LIN {X 0,Y 591.929,Z 246.123,A -85,B 0,C 180,E1 27050.152,E2 27050.152} C_VEL
LIN {X 0,Y 584.236,Z 228.435,A -85,B 0,C 180,E1 27048.26,E2 27048.26} C_VEL
LIN {X 0,Y 578.995,Z 217.335,A -85,B 0,C 180,E1 27047.073,E2 27047.073} C_VEL
LIN {X 0,Y 577.607,Z 214.744,A -85,B 0,C 180,E1 27046.785,E2 27046.785} C_VEL
LIN {X 0,Y 577.299,Z 213.311,A -85,B 0,C 180,E1 27046.634,E2 27046.634} C_VEL
LIN {X 0,Y 577.308,Z 213.309,A -85,B 0,C 180,E1 27043.304,E2 27043.304} C_VEL
LIN {X 0,Y 577.314,Z 213.308,A -85,B 0,C 180,E1 27040.046,E2 27040.046} C_VEL
LIN {X 0,Y 577.298,Z 213.305,A -85,B 0,C 180,E1 27036.818,E2 27036.818} C_VEL
LIN {X 0,Y 577.315,Z 213.304,A -85,B 0,C 180,E1 27033.539,E2 27033.539} C_VEL
LIN {X 0,Y 577.32,Z 213.314,A -85,B 0,C 180,E1 27030.15,E2 27030.15} C_VEL
LIN {X 0,Y 577.304,Z 213.311,A -85,B 0,C 180,E1 27026.876,E2 27026.876} C_VEL
LIN {X 0,Y 577.307,Z 213.291,A -85,B 0,C 180,E1 27023.584,E2 27023.584} C_VEL
LIN {X 0,Y 577.316,Z 213.314,A -85,B 0,C 180,E1 27020.267,E2 27020.267} C_VEL
LIN {X 0,Y 577.309,Z 213.299,A -85,B 0,C 180,E1 27016.916,E2 27016.916} C_VEL
LIN {X 0,Y 577.3,Z 213.303,A -85,B 0,C 180,E1 27013.674,E2 27013.674} C_VEL
LIN {X 0,Y 577.315,Z 213.307,A -85,B 0,C 180,E1 27010.341,E2 27010.341} C_VEL
LIN {X 0,Y 577.319,Z 213.3,A -85,B 0,C 180,E1 27006.964,E2 27006.964} C_VEL
LIN {X 0,Y 577.297,Z 213.318,A -85,B 0,C 180,E1 27003.674,E2 27003.674} C_VEL
LIN {X 0,Y 577.313,Z 213.295,A -85,B 0,C 180,E1 27000.397,E2 27000.397} C_VEL
LIN {X 0,Y 577.307,Z 213.312,A -85,B 0,C 180,E1 26997.121,E2 26997.121} C_VEL
LIN {X 0,Y 577.294,Z 213.294,A -85,B 0,C 180,E1 26993.818,E2 26993.818} C_VEL
LIN {X 0,Y 577.317,Z 213.31,A -85,B 0,C 180,E1 26990.53,E2 26990.53} C_VEL
LIN {X 0,Y 577.291,Z 213.316,A -85,B 0,C 180,E1 26987.293,E2 26987.293} C_VEL
LIN {X 0,Y 577.307,Z 213.316,A -85,B 0,C 180,E1 26983.999,E2 26983.999} C_VEL
LIN {X 0,Y 577.319,Z 213.312,A -85,B 0,C 180,E1 26980.682,E2 26980.682} C_VEL
LIN {X 0,Y 577.283,Z 213.322,A -85,B 0,C 180,E1 26977.494,E2 26977.494} C_VEL
LIN {X 0,Y 577.32,Z 213.321,A -85,B 0,C 180,E1 26974.232,E2 26974.232} C_VEL
LIN {X 0,Y 577.294,Z 213.316,A -85,B 0,C 180,E1 26970.989,E2 26970.989} C_VEL
LIN {X 0,Y 577.282,Z 213.322,A -85,B 0,C 180,E1 26967.642,E2 26967.642} C_VEL
LIN {X 0,Y 577.322,Z 213.313,A -85,B 0,C 180,E1 26964.413,E2 26964.413} C_VEL
LIN {X 0,Y 577.271,Z 213.322,A -85,B 0,C 180,E1 26961.21,E2 26961.21} C_VEL
LIN {X 0,Y 577.318,Z 213.515,A -85,B 0,C 180,E1 26960.825,E2 26960.825} C_VEL
LIN {X 0,Y 578.825,Z 217.068,A -85,B 0,C 180,E1 26960.399,E2 26960.399} C_VEL
LIN {X 0,Y 588.305,Z 235.653,A -85,B 0,C 180,E1 26958.091,E2 26958.091} C_VEL
LIN {X 0,Y 600.676,Z 260.638,A -85,B 0,C 180,E1 26955.24,E2 26955.24} C_VEL
LIN {X 0,Y 607.806,Z 275.644,A -85,B 0,C 180,E1 26953.662,E2 26953.662} C_VEL
LIN {X 0,Y 605.103,Z 308.798,A -85,B 0,C 180,E1 26951.828,E2 26951.828} C_VEL
LIN {X 0,Y 607.828,Z 331.376,A -85,B 0,C 180,E1 26951.271,E2 26951.271} C_VEL
LIN {X 0,Y 602.232,Z 577.23,A -85,B 0,C 180,E1 26947.881,E2 26947.881} C_VEL
LIN {X 0,Y 599.928,Z 692.589,A -85,B 0,C 180,E1 26946.326,E2 26946.326} C_VEL
LIN {X 0,Y 598.876,Z 717.126,A -85,B 0,C 180,E1 26945.833,E2 26945.833} C_VEL
LIN {X 0,Y 597.663,Z 738.821,A -85,B 0,C 180,E1 26945.256,E2 26945.256} C_VEL
LIN {X 0,Y 596.011,Z 763.246,A -85,B 0,C 180,E1 26944.428,E2 26944.428} C_VEL
LIN {X 0,Y 594.427,Z 783.289,A -85,B 0,C 180,E1 26943.601,E2 26943.601} C_VEL
LIN {X 0,Y 592.413,Z 806.84,A -85,B 0,C 180,E1 26942.444,E2 26942.444} C_VEL
LIN {X 0,Y 590.599,Z 826.305,A -85,B 0,C 180,E1 26941.316,E2 26941.316} C_VEL
LIN {X 0,Y 588.459,Z 848.134,A -85,B 0,C 180,E1 26939.858,E2 26939.858} C_VEL
LIN {X 0,Y 586.519,Z 867.008,A -85,B 0,C 180,E1 26938.397,E2 26938.397} C_VEL
LIN {X 0,Y 584.495,Z 887.006,A -85,B 0,C 180,E1 26936.628,E2 26936.628} C_VEL
LIN {X 0,Y 582.762,Z 903.916,A -85,B 0,C 180,E1 26934.912,E2 26934.912} C_VEL
LIN {X 0,Y 581.074,Z 921.418,A -85,B 0,C 180,E1 26932.886,E2 26932.886} C_VEL
LIN {X 0,Y 579.75,Z 935.465,A -85,B 0,C 180,E1 26931.023,E2 26931.023} C_VEL
LIN {X 0,Y 578.56,Z 949.769,A -85,B 0,C 180,E1 26928.855,E2 26928.855} C_VEL
LIN {X 0,Y 577.681,Z 961.419,A -85,B 0,C 180,E1 26926.801,E2 26926.801} C_VEL
LIN {X 0,Y 576.975,Z 972.466,A -85,B 0,C 180,E1 26924.553,E2 26924.553} C_VEL
LIN {X 0,Y 576.545,Z 980.188,A -85,B 0,C 180,E1 26922.622,E2 26922.622} C_VEL
LIN {X 0,Y 576.225,Z 987.119,A -85,B 0,C 180,E1 26920.498,E2 26920.498} C_VEL
LIN {X 0,Y 576.012,Z 993.449,A -85,B 0,C 180,E1 26918.083,E2 26918.083} C_VEL
LIN {X 0,Y 575.941,Z 997.697,A -85,B 0,C 180,E1 26915.852,E2 26915.852} C_VEL
LIN {X 0,Y 575.915,Z 1000.576,A -85,B 0,C 180,E1 26913.683,E2 26913.683} C_VEL
LIN {X 0,Y 575.907,Z 1002.235,A -85,B 0,C 180,E1 26911.194,E2 26911.194} C_VEL
LIN {X 0,Y 575.888,Z 1002.325,A -85,B 0,C 180,E1 26909.204,E2 26909.204} C_VEL
LIN {X 0,Y 575.886,Z 1001.289,A -85,B 0,C 180,E1 26907.114,E2 26907.114} C_VEL
LIN {X 0,Y 575.909,Z 998.45,A -85,B 0,C 180,E1 26904.62,E2 26904.62} C_VEL
LIN {X 0,Y 575.969,Z 994.688,A -85,B 0,C 180,E1 26902.519,E2 26902.519} C_VEL
LIN {X 0,Y 576.141,Z 989.457,A -85,B 0,C 180,E1 26900.308,E2 26900.308} C_VEL
LIN {X 0,Y 576.451,Z 981.951,A -85,B 0,C 180,E1 26897.884,E2 26897.884} C_VEL
LIN {X 0,Y 576.79,Z 975.298,A -85,B 0,C 180,E1 26896.117,E2 26896.117} C_VEL
LIN {X 0,Y 577.322,Z 966.57,A -85,B 0,C 180,E1 26894.222,E2 26894.222} C_VEL
LIN {X 0,Y 578.171,Z 954.305,A -85,B 0,C 180,E1 26891.967,E2 26891.967} C_VEL
LIN {X 0,Y 579.14,Z 941.931,A -85,B 0,C 180,E1 26890.01,E2 26890.01} C_VEL
LIN {X 0,Y 580.46,Z 926.019,A -85,B 0,C 180,E1 26887.837,E2 26887.837} C_VEL
LIN {X 0,Y 581.785,Z 911.136,A -85,B 0,C 180,E1 26886.071,E2 26886.071} C_VEL
LIN {X 0,Y 583.484,Z 892.287,A -85,B 0,C 180,E1 26884.115,E2 26884.115} C_VEL
LIN {X 0,Y 585.062,Z 875.137,A -85,B 0,C 180,E1 26882.568,E2 26882.568} C_VEL
LIN {X 0,Y 586.934,Z 854.247,A -85,B 0,C 180,E1 26880.92,E2 26880.92} C_VEL
LIN {X 0,Y 588.596,Z 834.717,A -85,B 0,C 180,E1 26879.587,E2 26879.587} C_VEL
LIN {X 0,Y 590.519,Z 811.335,A -85,B 0,C 180,E1 26878.213,E2 26878.213} C_VEL
LIN {X 0,Y 592.038,Z 790.551,A -85,B 0,C 180,E1 26877.171,E2 26877.171} C_VEL
LIN {X 0,Y 593.635,Z 766.597,A -85,B 0,C 180,E1 26876.168,E2 26876.168} C_VEL
LIN {X 0,Y 594.899,Z 744.933,A -85,B 0,C 180,E1 26875.42,E2 26875.42} C_VEL
LIN {X 0,Y 596.12,Z 719.728,A -85,B 0,C 180,E1 26874.739,E2 26874.739} C_VEL
LIN {X 0,Y 596.892,Z 698.83,A -85,B 0,C 180,E1 26874.312,E2 26874.312} C_VEL
LIN {X 0,Y 597.508,Z 665.557,A -85,B 0,C 180,E1 26873.847,E2 26873.847} C_VEL
LIN {X 0,Y 599.383,Z 523.368,A -85,B 0,C 180,E1 26872.041,E2 26872.041} C_VEL
LIN {X 0,Y 602.037,Z 398.059,A -85,B 0,C 180,E1 26870.281,E2 26870.281} C_VEL
LIN {X 0,Y 603.978,Z 328.15,A -85,B 0,C 180,E1 26869.204,E2 26869.204} C_VEL
LIN {X 0,Y 603.753,Z 324.587,A -85,B 0,C 180,E1 26869.08,E2 26869.08} C_VEL
LIN {X 0,Y 608.265,Z 300.685,A -85,B 0,C 180,E1 26867.429,E2 26867.429} C_VEL
LIN {X 0,Y 613.531,Z 280.646,A -85,B 0,C 180,E1 26865.901,E2 26865.901} C_VEL
LIN {X 0,Y 612.091,Z 275.219,A -85,B 0,C 180,E1 26864.716,E2 26864.716} C_VEL
LIN {X 0,Y 611.11,Z 271.585,A -85,B 0,C 180,E1 26863.538,E2 26863.538} C_VEL
LIN {X 0,Y 610.691,Z 269.324,A -85,B 0,C 180,E1 26862.123,E2 26862.123} C_VEL
LIN {X 0,Y 610.625,Z 269.272,A -85,B 0,C 180,E1 26861.543,E2 26861.543} C_VEL
LIN {X 0,Y 610.726,Z 271.372,A -85,B 0,C 180,E1 26860.048,E2 26860.048} C_VEL
LIN {X 0,Y 611.329,Z 275.332,A -85,B 0,C 180,E1 26858.788,E2 26858.788} C_VEL
LIN {X 0,Y 611.672,Z 278.803,A -85,B 0,C 180,E1 26858.045,E2 26858.045} C_VEL
LIN {X 0,Y 605.574,Z 300.252,A -85,B 0,C 180,E1 26856.119,E2 26856.119} C_VEL
LIN {X 0,Y 599.965,Z 327.92,A -85,B 0,C 180,E1 26853.824,E2 26853.824} C_VEL
LIN {X 0,Y 595.013,Z 362.924,A -85,B 0,C 180,E1 26851.114,E2 26851.114} C_VEL
LIN {X 0,Y 590.47,Z 407.602,A -85,B 0,C 180,E1 26847.878,E2 26847.878} C_VEL
LIN {X 0,Y 589.4,Z 422.994,A -85,B 0,C 180,E1 26846.832,E2 26846.832} C_VEL
LIN {X 0,Y 592.686,Z 455.008,A -85,B 0,C 180,E1 26845.661,E2 26845.661} C_VEL
LIN {X 0,Y 595.543,Z 491.146,A -85,B 0,C 180,E1 26844.524,E2 26844.524} C_VEL
LIN {X 0,Y 594.867,Z 505.645,A -85,B 0,C 180,E1 26844.22,E2 26844.22} C_VEL
LIN {X 0,Y 589.455,Z 607.464,A -85,B 0,C 180,E1 26842.27,E2 26842.27} C_VEL
LIN {X 0,Y 586.293,Z 687.572,A -85,B 0,C 180,E1 26840.777,E2 26840.777} C_VEL
LIN {X 0,Y 585.33,Z 709.905,A -85,B 0,C 180,E1 26840.167,E2 26840.167} C_VEL
LIN {X 0,Y 584.359,Z 731.272,A -85,B 0,C 180,E1 26839.387,E2 26839.387} C_VEL
LIN {X 0,Y 583.386,Z 750.706,A -85,B 0,C 180,E1 26838.486,E2 26838.486} C_VEL
LIN {X 0,Y 582.433,Z 769.003,A -85,B 0,C 180,E1 26837.432,E2 26837.432} C_VEL
LIN {X 0,Y 581.473,Z 786.178,A -85,B 0,C 180,E1 26836.226,E2 26836.226} C_VEL
LIN {X 0,Y 580.594,Z 801.262,A -85,B 0,C 180,E1 26834.951,E2 26834.951} C_VEL
LIN {X 0,Y 579.773,Z 814.876,A -85,B 0,C 180,E1 26833.565,E2 26833.565} C_VEL
LIN {X 0,Y 579.038,Z 827.147,A -85,B 0,C 180,E1 26832.061,E2 26832.061} C_VEL
LIN {X 0,Y 578.439,Z 837.273,A -85,B 0,C 180,E1 26830.558,E2 26830.558} C_VEL
LIN {X 0,Y 577.896,Z 846.496,A -85,B 0,C 180,E1 26828.858,E2 26828.858} C_VEL
LIN {X 0,Y 577.499,Z 853.707,A -85,B 0,C 180,E1 26827.161,E2 26827.161} C_VEL
LIN {X 0,Y 577.21,Z 859.389,A -85,B 0,C 180,E1 26825.368,E2 26825.368} C_VEL
LIN {X 0,Y 576.993,Z 863.232,A -85,B 0,C 180,E1 26823.577,E2 26823.577} C_VEL
LIN {X 0,Y 576.852,Z 865.342,A -85,B 0,C 180,E1 26821.788,E2 26821.788} C_VEL
LIN {X 0,Y 576.771,Z 865.736,A -85,B 0,C 180,E1 26819.901,E2 26819.901} C_VEL
LIN {X 0,Y 576.736,Z 864.293,A -85,B 0,C 180,E1 26818.013,E2 26818.013} C_VEL
LIN {X 0,Y 576.764,Z 861.014,A -85,B 0,C 180,E1 26816.123,E2 26816.123} C_VEL
LIN {X 0,Y 576.874,Z 856.161,A -85,B 0,C 180,E1 26814.33,E2 26814.33} C_VEL
LIN {X 0,Y 577.061,Z 849.471,A -85,B 0,C 180,E1 26812.533,E2 26812.533} C_VEL
LIN {X 0,Y 577.367,Z 841.126,A -85,B 0,C 180,E1 26810.799,E2 26810.799} C_VEL
LIN {X 0,Y 577.814,Z 831.101,A -85,B 0,C 180,E1 26809.128,E2 26809.128} C_VEL
LIN {X 0,Y 578.397,Z 819.329,A -85,B 0,C 180,E1 26807.52,E2 26807.52} C_VEL
LIN {X 0,Y 579.11,Z 805.98,A -85,B 0,C 180,E1 26806.012,E2 26806.012} C_VEL
LIN {X 0,Y 579.937,Z 790.987,A -85,B 0,C 180,E1 26804.602,E2 26804.602} C_VEL
LIN {X 0,Y 580.827,Z 774.875,A -85,B 0,C 180,E1 26803.344,E2 26803.344} C_VEL
LIN {X 0,Y 581.733,Z 757.436,A -85,B 0,C 180,E1 26802.218,E2 26802.218} C_VEL
LIN {X 0,Y 582.635,Z 739.626,A -85,B 0,C 180,E1 26801.281,E2 26801.281} C_VEL
LIN {X 0,Y 583.514,Z 720.275,A -85,B 0,C 180,E1 26800.469,E2 26800.469} C_VEL
LIN {X 0,Y 584.279,Z 700.12,A -85,B 0,C 180,E1 26799.828,E2 26799.828} C_VEL
LIN {X 0,Y 584.919,Z 679.428,A -85,B 0,C 180,E1 26799.37,E2 26799.37} C_VEL
LIN {X 0,Y 588.981,Z 489.215,A -85,B 0,C 180,E1 26796.534,E2 26796.534} C_VEL
LIN {X 0,Y 585.221,Z 455.543,A -85,B 0,C 180,E1 26795.791,E2 26795.791} C_VEL
LIN {X 0,Y 587.587,Z 405.605,A -85,B 0,C 180,E1 26792.594,E2 26792.594} C_VEL
LIN {X 0,Y 590.441,Z 352.546,A -85,B 0,C 180,E1 26789.158,E2 26789.158} C_VEL
LIN {X 0,Y 593.46,Z 300.77,A -85,B 0,C 180,E1 26785.754,E2 26785.754} C_VEL
LIN {X 0,Y 595.914,Z 261.134,A -85,B 0,C 180,E1 26783.108,E2 26783.108} C_VEL
LIN {X 0,Y 591.877,Z 250.242,A -85,B 0,C 180,E1 26782.056,E2 26782.056} C_VEL
LIN {X 0,Y 589.101,Z 245.546,A -85,B 0,C 180,E1 26781.522,E2 26781.522} C_VEL
LIN {X 0,Y 577.793,Z 233.961,A -85,B 0,C 180,E1 26779.852,E2 26779.852} C_VEL
LIN {X 0,Y 576.198,Z 231.311,A -85,B 0,C 180,E1 26779.532,E2 26779.532} C_VEL
LIN {X 0,Y 569.344,Z 214.421,A -85,B 0,C 180,E1 26777.698,E2 26777.698} C_VEL
LIN {X 0,Y 569.381,Z 214.302,A -85,B 0,C 180,E1 26774.482,E2 26774.482} C_VEL
LIN {X 0,Y 569.39,Z 214.435,A -85,B 0,C 180,E1 26773.881,E2 26773.881} C_VEL
LIN {X 0,Y 570.341,Z 217.235,A -85,B 0,C 180,E1 26773.61,E2 26773.61} C_VEL
LIN {X 0,Y 571.71,Z 219.791,A -85,B 0,C 180,E1 26773.317,E2 26773.317} C_VEL
LIN {X 0,Y 578.876,Z 234.711,A -85,B 0,C 180,E1 26771.683,E2 26771.683} C_VEL
LIN {X 0,Y 586.838,Z 253.704,A -85,B 0,C 180,E1 26769.633,E2 26769.633} C_VEL
LIN {X 0,Y 593.746,Z 272.147,A -85,B 0,C 180,E1 26767.674,E2 26767.674} C_VEL
LIN {X 0,Y 592.76,Z 314.667,A -85,B 0,C 180,E1 26764.643,E2 26764.643} C_VEL
LIN {X 0,Y 592.824,Z 338.961,A -85,B 0,C 180,E1 26763.068,E2 26763.068} C_VEL
LIN {X 0,Y 591.933,Z 343.747,A -85,B 0,C 180,E1 26762.899,E2 26762.899} C_VEL
LIN {X 0,Y 589.728,Z 439.794,A -85,B 0,C 180,E1 26761.581,E2 26761.581} C_VEL
LIN {X 0,Y 586.74,Z 530.066,A -85,B 0,C 180,E1 26760.163,E2 26760.163} C_VEL
LIN {X 0,Y 583.259,Z 625.148,A -85,B 0,C 180,E1 26758.492,E2 26758.492} C_VEL
LIN {X 0,Y 582.489,Z 647.168,A -85,B 0,C 180,E1 26757.952,E2 26757.952} C_VEL
LIN {X 0,Y 581.453,Z 668.771,A -85,B 0,C 180,E1 26757.245,E2 26757.245} C_VEL
LIN {X 0,Y 580.207,Z 690.159,A -85,B 0,C 180,E1 26756.345,E2 26756.345} C_VEL
LIN {X 0,Y 578.823,Z 710.131,A -85,B 0,C 180,E1 26755.312,E2 26755.312} C_VEL
LIN {X 0,Y 577.378,Z 729.317,A -85,B 0,C 180,E1 26754.123,E2 26754.123} C_VEL
LIN {X 0,Y 575.82,Z 748.322,A -85,B 0,C 180,E1 26752.728,E2 26752.728} C_VEL
LIN {X 0,Y 574.417,Z 765.121,A -85,B 0,C 180,E1 26751.281,E2 26751.281} C_VEL
LIN {X 0,Y 573.057,Z 781.033,A -85,B 0,C 180,E1 26749.679,E2 26749.679} C_VEL
LIN {X 0,Y 571.809,Z 795.88,A -85,B 0,C 180,E1 26747.924,E2 26747.924} C_VEL
LIN {X 0,Y 570.757,Z 809.256,A -85,B 0,C 180,E1 26746.069,E2 26746.069} C_VEL
LIN {X 0,Y 569.863,Z 821.736,A -85,B 0,C 180,E1 26744.013,E2 26744.013} C_VEL
LIN {X 0,Y 569.248,Z 831.607,A -85,B 0,C 180,E1 26742.065,E2 26742.065} C_VEL
LIN {X 0,Y 568.806,Z 840.094,A -85,B 0,C 180,E1 26740.022,E2 26740.022} C_VEL
LIN {X 0,Y 568.521,Z 846.753,A -85,B 0,C 180,E1 26737.987,E2 26737.987} C_VEL
LIN {X 0,Y 568.361,Z 852.257,A -85,B 0,C 180,E1 26735.755,E2 26735.755} C_VEL
LIN {X 0,Y 568.297,Z 855.835,A -85,B 0,C 180,E1 26733.632,E2 26733.632} C_VEL
LIN {X 0,Y 568.26,Z 857.744,A -85,B 0,C 180,E1 26731.512,E2 26731.512} C_VEL
LIN {X 0,Y 568.247,Z 858.093,A -85,B 0,C 180,E1 26729.395,E2 26729.395} C_VEL
LIN {X 0,Y 568.274,Z 856.938,A -85,B 0,C 180,E1 26727.277,E2 26727.277} C_VEL
LIN {X 0,Y 568.33,Z 854.144,A -85,B 0,C 180,E1 26725.156,E2 26725.156} C_VEL
LIN {X 0,Y 568.421,Z 849.713,A -85,B 0,C 180,E1 26723.029,E2 26723.029} C_VEL
LIN {X 0,Y 568.641,Z 843.588,A -85,B 0,C 180,E1 26720.894,E2 26720.894} C_VEL
LIN {X 0,Y 569.027,Z 836.048,A -85,B 0,C 180,E1 26718.855,E2 26718.855} C_VEL
LIN {X 0,Y 569.547,Z 826.578,A -85,B 0,C 180,E1 26716.807,E2 26716.807} C_VEL
LIN {X 0,Y 570.279,Z 815.707,A -85,B 0,C 180,E1 26714.856,E2 26714.856} C_VEL
LIN {X 0,Y 571.203,Z 803.495,A -85,B 0,C 180,E1 26713.002,E2 26713.002} C_VEL
LIN {X 0,Y 572.319,Z 789.976,A -85,B 0,C 180,E1 26711.249,E2 26711.249} C_VEL
LIN {X 0,Y 573.661,Z 774.003,A -85,B 0,C 180,E1 26709.492,E2 26709.492} C_VEL
LIN {X 0,Y 575.071,Z 757.356,A -85,B 0,C 180,E1 26707.933,E2 26707.933} C_VEL
LIN {X 0,Y 576.568,Z 739.348,A -85,B 0,C 180,E1 26706.493,E2 26706.493} C_VEL
LIN {X 0,Y 578.148,Z 719.445,A -85,B 0,C 180,E1 26705.149,E2 26705.149} C_VEL
LIN {X 0,Y 579.515,Z 700.296,A -85,B 0,C 180,E1 26704.063,E2 26704.063} C_VEL
LIN {X 0,Y 580.878,Z 679.328,A -85,B 0,C 180,E1 26703.082,E2 26703.082} C_VEL
LIN {X 0,Y 581.989,Z 658.553,A -85,B 0,C 180,E1 26702.307,E2 26702.307} C_VEL
LIN {X 0,Y 582.878,Z 636.878,A -85,B 0,C 180,E1 26701.682,E2 26701.682} C_VEL
LIN {X 0,Y 583.753,Z 609.709,A -85,B 0,C 180,E1 26701.124,E2 26701.124} C_VEL
LIN {X 0,Y 587.697,Z 503.594,A -85,B 0,C 180,E1 26699.312,E2 26699.312} C_VEL
LIN {X 0,Y 590.36,Z 417.842,A -85,B 0,C 180,E1 26698.011,E2 26698.011} C_VEL
LIN {X 0,Y 591.983,Z 342.833,A -85,B 0,C 180,E1 26696.995,E2 26696.995} C_VEL
LIN {X 0,Y 592.926,Z 337.654,A -85,B 0,C 180,E1 26696.765,E2 26696.765} C_VEL
LIN {X 0,Y 592.875,Z 307.651,A -85,B 0,C 180,E1 26694.775,E2 26694.775} C_VEL
LIN {X 0,Y 593.748,Z 271.834,A -85,B 0,C 180,E1 26692.194,E2 26692.194} C_VEL
LIN {X 0,Y 585.364,Z 249.888,A -85,B 0,C 180,E1 26689.854,E2 26689.854} C_VEL
LIN {X 0,Y 578.158,Z 233.181,A -85,B 0,C 180,E1 26688.044,E2 26688.044} C_VEL
LIN {X 0,Y 571.21,Z 218.485,A -85,B 0,C 180,E1 26686.444,E2 26686.444} C_VEL
LIN {X 0,Y 569.605,Z 215.436,A -85,B 0,C 180,E1 26686.101,E2 26686.101} C_VEL
LIN {X 0,Y 569.377,Z 214.299,A -85,B 0,C 180,E1 26685.974,E2 26685.974} C_VEL
LIN {X 0,Y 569.36,Z 214.306,A -85,B 0,C 180,E1 26682.678,E2 26682.678} C_VEL
LIN {X 0,Y 569.378,Z 214.305,A -85,B 0,C 180,E1 26679.343,E2 26679.343} C_VEL
LIN {X 0,Y 569.374,Z 214.297,A -85,B 0,C 180,E1 26676.037,E2 26676.037} C_VEL
LIN {X 0,Y 569.361,Z 214.289,A -85,B 0,C 180,E1 26672.733,E2 26672.733} C_VEL
LIN {X 0,Y 569.38,Z 214.295,A -85,B 0,C 180,E1 26669.422,E2 26669.422} C_VEL
LIN {X 0,Y 569.374,Z 214.308,A -85,B 0,C 180,E1 26666.042,E2 26666.042} C_VEL
LIN {X 0,Y 569.365,Z 214.284,A -85,B 0,C 180,E1 26662.728,E2 26662.728} C_VEL
LIN {X 0,Y 569.371,Z 214.293,A -85,B 0,C 180,E1 26659.431,E2 26659.431} C_VEL
LIN {X 0,Y 569.372,Z 214.303,A -85,B 0,C 180,E1 26656.005,E2 26656.005} C_VEL
LIN {X 0,Y 569.369,Z 214.281,A -85,B 0,C 180,E1 26652.784,E2 26652.784} C_VEL
LIN {X 0,Y 569.363,Z 214.305,A -85,B 0,C 180,E1 26649.502,E2 26649.502} C_VEL
LIN {X 0,Y 569.374,Z 214.277,A -85,B 0,C 180,E1 26646.15,E2 26646.15} C_VEL
LIN {X 0,Y 569.376,Z 214.304,A -85,B 0,C 180,E1 26642.818,E2 26642.818} C_VEL
LIN {X 0,Y 569.352,Z 214.275,A -85,B 0,C 180,E1 26639.598,E2 26639.598} C_VEL
LIN {X 0,Y 569.376,Z 214.308,A -85,B 0,C 180,E1 26636.275,E2 26636.275} C_VEL
LIN {X 0,Y 569.38,Z 214.272,A -85,B 0,C 180,E1 26632.939,E2 26632.939} C_VEL
LIN {X 0,Y 569.35,Z 214.308,A -85,B 0,C 180,E1 26629.578,E2 26629.578} C_VEL
LIN {X 0,Y 569.382,Z 214.308,A -85,B 0,C 180,E1 26626.286,E2 26626.286} C_VEL
LIN {X 0,Y 569.361,Z 214.306,A -85,B 0,C 180,E1 26623.051,E2 26623.051} C_VEL
LIN {X 0,Y 569.348,Z 214.308,A -85,B 0,C 180,E1 26619.651,E2 26619.651} C_VEL
LIN {X 0,Y 569.383,Z 214.305,A -85,B 0,C 180,E1 26616.397,E2 26616.397} C_VEL
LIN {X 0,Y 569.346,Z 214.301,A -85,B 0,C 180,E1 26613.145,E2 26613.145} C_VEL
LIN {X 0,Y 569.353,Z 214.312,A -85,B 0,C 180,E1 26609.774,E2 26609.774} C_VEL
LIN {X 0,Y 569.381,Z 214.303,A -85,B 0,C 180,E1 26606.527,E2 26606.527} C_VEL
LIN {X 0,Y 569.334,Z 214.309,A -85,B 0,C 180,E1 26603.336,E2 26603.336} C_VEL
LIN {X 0,Y 569.358,Z 214.444,A -85,B 0,C 180,E1 26601.594,E2 26601.594} C_VEL
LIN {X 0,Y 570.387,Z 217.397,A -85,B 0,C 180,E1 26601.257,E2 26601.257} C_VEL
LIN {X 0,Y 571.764,Z 219.658,A -85,B 0,C 180,E1 26600.937,E2 26600.937} C_VEL
LIN {X 0,Y 581.042,Z 238.068,A -85,B 0,C 180,E1 26598.616,E2 26598.616} C_VEL
LIN {X 0,Y 592.456,Z 260.848,A -85,B 0,C 180,E1 26595.946,E2 26595.946} C_VEL
LIN {X 0,Y 601.171,Z 279.402,A -85,B 0,C 180,E1 26593.964,E2 26593.964} C_VEL
LIN {X 0,Y 598.614,Z 309.394,A -85,B 0,C 180,E1 26592.29,E2 26592.29} C_VEL
LIN {X 0,Y 601.382,Z 332.717,A -85,B 0,C 180,E1 26591.709,E2 26591.709} C_VEL
LIN {X 0,Y 595.541,Z 572.332,A -85,B 0,C 180,E1 26588.354,E2 26588.354} C_VEL
LIN {X 0,Y 592.986,Z 692.835,A -85,B 0,C 180,E1 26586.707,E2 26586.707} C_VEL
LIN {X 0,Y 591.882,Z 717.267,A -85,B 0,C 180,E1 26586.21,E2 26586.21} C_VEL
LIN {X 0,Y 590.638,Z 738.58,A -85,B 0,C 180,E1 26585.637,E2 26585.637} C_VEL
LIN {X 0,Y 588.881,Z 763.35,A -85,B 0,C 180,E1 26584.786,E2 26584.786} C_VEL
LIN {X 0,Y 587.231,Z 783.315,A -85,B 0,C 180,E1 26583.952,E2 26583.952} C_VEL
LIN {X 0,Y 585.054,Z 807.455,A -85,B 0,C 180,E1 26582.746,E2 26582.746} C_VEL
LIN {X 0,Y 583.145,Z 827.122,A -85,B 0,C 180,E1 26581.589,E2 26581.589} C_VEL
LIN {X 0,Y 580.833,Z 849.426,A -85,B 0,C 180,E1 26580.063,E2 26580.063} C_VEL
LIN {X 0,Y 578.942,Z 867.051,A -85,B 0,C 180,E1 26578.673,E2 26578.673} C_VEL
LIN {X 0,Y 576.775,Z 887.323,A -85,B 0,C 180,E1 26576.846,E2 26576.846} C_VEL
LIN {X 0,Y 575.028,Z 903.654,A -85,B 0,C 180,E1 26575.16,E2 26575.16} C_VEL
LIN {X 0,Y 573.254,Z 921.098,A -85,B 0,C 180,E1 26573.107,E2 26573.107} C_VEL
LIN {X 0,Y 571.882,Z 935.11,A -85,B 0,C 180,E1 26571.218,E2 26571.218} C_VEL
LIN {X 0,Y 570.586,Z 949.964,A -85,B 0,C 180,E1 26568.917,E2 26568.917} C_VEL
LIN {X 0,Y 569.728,Z 960.976,A -85,B 0,C 180,E1 26566.938,E2 26566.938} C_VEL
LIN {X 0,Y 568.973,Z 972.391,A -85,B 0,C 180,E1 26564.555,E2 26564.555} C_VEL
LIN {X 0,Y 568.499,Z 980.992,A -85,B 0,C 180,E1 26562.391,E2 26562.391} C_VEL
LIN {X 0,Y 568.169,Z 988.802,A -85,B 0,C 180,E1 26560.033,E2 26560.033} C_VEL
LIN {X 0,Y 567.986,Z 994.275,A -85,B 0,C 180,E1 26557.79,E2 26557.79} C_VEL
LIN {X 0,Y 567.934,Z 997.972,A -85,B 0,C 180,E1 26555.759,E2 26555.759} C_VEL
LIN {X 0,Y 567.903,Z 1001.015,A -85,B 0,C 180,E1 26553.331,E2 26553.331} C_VEL
LIN {X 0,Y 567.898,Z 1002.28,A -85,B 0,C 180,E1 26551.009,E2 26551.009} C_VEL
LIN {X 0,Y 567.898,Z 1002.28,A -85,B 0,C 180,E1 26548.991,E2 26548.991} C_VEL
LIN {X 0,Y 567.906,Z 1000.915,A -85,B 0,C 180,E1 26546.568,E2 26546.568} C_VEL
LIN {X 0,Y 567.934,Z 997.971,A -85,B 0,C 180,E1 26544.24,E2 26544.24} C_VEL
LIN {X 0,Y 567.993,Z 994.069,A -85,B 0,C 180,E1 26542.108,E2 26542.108} C_VEL
LIN {X 0,Y 568.191,Z 988.158,A -85,B 0,C 180,E1 26539.762,E2 26539.762} C_VEL
LIN {X 0,Y 568.5,Z 980.91,A -85,B 0,C 180,E1 26537.609,E2 26537.609} C_VEL
LIN {X 0,Y 568.978,Z 972.186,A -85,B 0,C 180,E1 26535.445,E2 26535.445} C_VEL
LIN {X 0,Y 569.688,Z 961.092,A -85,B 0,C 180,E1 26533.166,E2 26533.166} C_VEL
LIN {X 0,Y 570.533,Z 949.674,A -85,B 0,C 180,E1 26531.153,E2 26531.153} C_VEL
LIN {X 0,Y 571.694,Z 935.436,A -85,B 0,C 180,E1 26528.989,E2 26528.989} C_VEL
LIN {X 0,Y 572.997,Z 921.077,A -85,B 0,C 180,E1 26527.099,E2 26527.099} C_VEL
LIN {X 0,Y 574.602,Z 903.659,A -85,B 0,C 180,E1 26525.095,E2 26525.095} C_VEL
LIN {X 0,Y 576.157,Z 887.303,A -85,B 0,C 180,E1 26523.456,E2 26523.456} C_VEL
LIN {X 0,Y 577.957,Z 868.083,A -85,B 0,C 180,E1 26521.76,E2 26521.76} C_VEL
LIN {X 0,Y 579.754,Z 848.643,A -85,B 0,C 180,E1 26520.274,E2 26520.274} C_VEL
LIN {X 0,Y 581.774,Z 826.231,A -85,B 0,C 180,E1 26518.789,E2 26518.789} C_VEL
LIN {X 0,Y 583.371,Z 806.617,A -85,B 0,C 180,E1 26517.672,E2 26517.672} C_VEL
LIN {X 0,Y 585.213,Z 782.574,A -85,B 0,C 180,E1 26516.504,E2 26516.504} C_VEL
LIN {X 0,Y 586.653,Z 761.498,A -85,B 0,C 180,E1 26515.656,E2 26515.656} C_VEL
LIN {X 0,Y 588.125,Z 736.578,A -85,B 0,C 180,E1 26514.836,E2 26514.836} C_VEL
LIN {X 0,Y 589.14,Z 714.548,A -85,B 0,C 180,E1 26514.274,E2 26514.274} C_VEL
LIN {X 0,Y 590.03,Z 688.498,A -85,B 0,C 180,E1 26513.789,E2 26513.789} C_VEL
LIN {X 0,Y 592.517,Z 526.417,A -85,B 0,C 180,E1 26511.677,E2 26511.677} C_VEL
LIN {X 0,Y 595.353,Z 407.844,A -85,B 0,C 180,E1 26509.964,E2 26509.964} C_VEL
LIN {X 0,Y 597.915,Z 329.601,A -85,B 0,C 180,E1 26508.72,E2 26508.72} C_VEL
LIN {X 0,Y 597.763,Z 327.352,A -85,B 0,C 180,E1 26508.645,E2 26508.645} C_VEL
LIN {X 0,Y 602.798,Z 303.687,A -85,B 0,C 180,E1 26506.955,E2 26506.955} C_VEL
LIN {X 0,Y 608.154,Z 285.464,A -85,B 0,C 180,E1 26505.525,E2 26505.525} C_VEL
LIN {X 0,Y 607.008,Z 280.361,A -85,B 0,C 180,E1 26504.302,E2 26504.302} C_VEL
LIN {X 0,Y 606.272,Z 277.736,A -85,B 0,C 180,E1 26503.321,E2 26503.321} C_VEL
LIN {X 0,Y 606.126,Z 275.632,A -85,B 0,C 180,E1 26501.786,E2 26501.786} C_VEL
LIN {X 0,Y 605.897,Z 277.499,A -85,B 0,C 180,E1 26500.309,E2 26500.309} C_VEL
LIN {X 0,Y 606.251,Z 280.584,A -85,B 0,C 180,E1 26499.175,E2 26499.175} C_VEL
LIN {X 0,Y 606.491,Z 283.655,A -85,B 0,C 180,E1 26498.429,E2 26498.429} C_VEL
LIN {X 0,Y 599.82,Z 304.959,A -85,B 0,C 180,E1 26496.462,E2 26496.462} C_VEL
LIN {X 0,Y 593.809,Z 331.937,A -85,B 0,C 180,E1 26494.164,E2 26494.164} C_VEL
LIN {X 0,Y 588.656,Z 364.932,A -85,B 0,C 180,E1 26491.545,E2 26491.545} C_VEL
LIN {X 0,Y 583.914,Z 406.935,A -85,B 0,C 180,E1 26488.428,E2 26488.428} C_VEL
LIN {X 0,Y 582.884,Z 419.506,A -85,B 0,C 180,E1 26487.553,E2 26487.553} C_VEL
LIN {X 0,Y 585.632,Z 446.596,A -85,B 0,C 180,E1 26486.495,E2 26486.495} C_VEL
LIN {X 0,Y 588.405,Z 481.333,A -85,B 0,C 180,E1 26485.31,E2 26485.31} C_VEL
LIN {X 0,Y 589.088,Z 495.815,A -85,B 0,C 180,E1 26484.884,E2 26484.884} C_VEL
LIN {X 0,Y 583.019,Z 598.12,A -85,B 0,C 180,E1 26482.848,E2 26482.848} C_VEL
LIN {X 0,Y 579.118,Z 687.482,A -85,B 0,C 180,E1 26481.13,E2 26481.13} C_VEL
LIN {X 0,Y 578.059,Z 710.48,A -85,B 0,C 180,E1 26480.491,E2 26480.491} C_VEL
LIN {X 0,Y 577.073,Z 730.613,A -85,B 0,C 180,E1 26479.748,E2 26479.748} C_VEL
LIN {X 0,Y 576.021,Z 750.164,A -85,B 0,C 180,E1 26478.837,E2 26478.837} C_VEL
LIN {X 0,Y 575.015,Z 768.532,A -85,B 0,C 180,E1 26477.785,E2 26477.785} C_VEL
LIN {X 0,Y 574.02,Z 785.524,A -85,B 0,C 180,E1 26476.599,E2 26476.599} C_VEL
LIN {X 0,Y 573.042,Z 801.208,A -85,B 0,C 180,E1 26475.277,E2 26475.277} C_VEL
LIN {X 0,Y 572.151,Z 815.237,A -85,B 0,C 180,E1 26473.852,E2 26473.852} C_VEL
LIN {X 0,Y 571.352,Z 827.64,A -85,B 0,C 180,E1 26472.328,E2 26472.328} C_VEL
LIN {X 0,Y 570.654,Z 838.462,A -85,B 0,C 180,E1 26470.704,E2 26470.704} C_VEL
LIN {X 0,Y 570.107,Z 847.239,A -85,B 0,C 180,E1 26469.082,E2 26469.082} C_VEL
LIN {X 0,Y 569.668,Z 854.55,A -85,B 0,C 180,E1 26467.362,E2 26467.362} C_VEL
LIN {X 0,Y 569.345,Z 860.304,A -85,B 0,C 180,E1 26465.543,E2 26465.543} C_VEL
LIN {X 0,Y 569.089,Z 864.343,A -85,B 0,C 180,E1 26463.643,E2 26463.643} C_VEL
LIN {X 0,Y 568.932,Z 866.445,A -85,B 0,C 180,E1 26461.813,E2 26461.813} C_VEL
LIN {X 0,Y 568.841,Z 866.79,A -85,B 0,C 180,E1 26459.899,E2 26459.899} C_VEL
LIN {X 0,Y 568.802,Z 865.285,A -85,B 0,C 180,E1 26457.985,E2 26457.985} C_VEL
LIN {X 0,Y 568.828,Z 862.171,A -85,B 0,C 180,E1 26456.17,E2 26456.17} C_VEL
LIN {X 0,Y 568.939,Z 857.335,A -85,B 0,C 180,E1 26454.352,E2 26454.352} C_VEL
LIN {X 0,Y 569.132,Z 850.663,A -85,B 0,C 180,E1 26452.53,E2 26452.53} C_VEL
LIN {X 0,Y 569.443,Z 842.522,A -85,B 0,C 180,E1 26450.805,E2 26450.805} C_VEL
LIN {X 0,Y 569.912,Z 832.342,A -85,B 0,C 180,E1 26449.077,E2 26449.077} C_VEL
LIN {X 0,Y 570.518,Z 820.608,A -85,B 0,C 180,E1 26447.448,E2 26447.448} C_VEL
LIN {X 0,Y 571.257,Z 807.31,A -85,B 0,C 180,E1 26445.919,E2 26445.919} C_VEL
LIN {X 0,Y 572.113,Z 792.39,A -85,B 0,C 180,E1 26444.49,E2 26444.49} C_VEL
LIN {X 0,Y 573.037,Z 776.385,A -85,B 0,C 180,E1 26443.215,E2 26443.215} C_VEL
LIN {X 0,Y 573.957,Z 759.406,A -85,B 0,C 180,E1 26442.092,E2 26442.092} C_VEL
LIN {X 0,Y 574.926,Z 741.101,A -85,B 0,C 180,E1 26441.104,E2 26441.104} C_VEL
LIN {X 0,Y 575.801,Z 722.815,A -85,B 0,C 180,E1 26440.313,E2 26440.313} C_VEL
LIN {X 0,Y 576.605,Z 703.153,A -85,B 0,C 180,E1 26439.654,E2 26439.654} C_VEL
LIN {X 0,Y 577.304,Z 682.763,A -85,B 0,C 180,E1 26439.163,E2 26439.163} C_VEL
LIN {X 0,Y 581.678,Z 489.866,A -85,B 0,C 180,E1 26436.211,E2 26436.211} C_VEL
LIN {X 0,Y 577.785,Z 454.855,A -85,B 0,C 180,E1 26435.432,E2 26435.432} C_VEL
LIN {X 0,Y 580.371,Z 403.516,A -85,B 0,C 180,E1 26432.107,E2 26432.107} C_VEL
LIN {X 0,Y 583.308,Z 351.623,A -85,B 0,C 180,E1 26428.708,E2 26428.708} C_VEL
LIN {X 0,Y 586.526,Z 299.648,A -85,B 0,C 180,E1 26425.255,E2 26425.255} C_VEL
LIN {X 0,Y 588.85,Z 264.23,A -85,B 0,C 180,E1 26422.867,E2 26422.867} C_VEL
LIN {X 0,Y 580.082,Z 241.04,A -85,B 0,C 180,E1 26420.554,E2 26420.554} C_VEL
LIN {X 0,Y 576.198,Z 231.311,A -85,B 0,C 180,E1 26419.532,E2 26419.532} C_VEL
LIN {X 0,Y 573.888,Z 228.587,A -85,B 0,C 180,E1 26419.15,E2 26419.15} C_VEL
LIN {X 0,Y 565.359,Z 223.504,A -85,B 0,C 180,E1 26418.095,E2 26418.095} C_VEL
LIN {X 0,Y 563.532,Z 221.076,A -85,B 0,C 180,E1 26417.76,E2 26417.76} C_VEL
LIN {X 0,Y 561.425,Z 215.295,A -85,B 0,C 180,E1 26417.095,E2 26417.095} C_VEL
LIN {X 0,Y 561.47,Z 215.494,A -85,B 0,C 180,E1 26414.56,E2 26414.56} C_VEL
LIN {X 0,Y 562.583,Z 218.532,A -85,B 0,C 180,E1 26414.253,E2 26414.253} C_VEL
LIN {X 0,Y 563.947,Z 221.073,A -85,B 0,C 180,E1 26413.958,E2 26413.958} C_VEL
LIN {X 0,Y 571.17,Z 235.872,A -85,B 0,C 180,E1 26412.3,E2 26412.3} C_VEL
LIN {X 0,Y 578.648,Z 253.223,A -85,B 0,C 180,E1 26410.39,E2 26410.39} C_VEL
LIN {X 0,Y 587.03,Z 275.288,A -85,B 0,C 180,E1 26408.021,E2 26408.021} C_VEL
LIN {X 0,Y 586.494,Z 302.823,A -85,B 0,C 180,E1 26406.028,E2 26406.028} C_VEL
LIN {X 0,Y 586.337,Z 334.407,A -85,B 0,C 180,E1 26403.893,E2 26403.893} C_VEL
LIN {X 0,Y 586.342,Z 340.65,A -85,B 0,C 180,E1 26403.508,E2 26403.508} C_VEL
LIN {X 0,Y 585.23,Z 346.433,A -85,B 0,C 180,E1 26403.299,E2 26403.299} C_VEL
LIN {X 0,Y 582.959,Z 441.18,A -85,B 0,C 180,E1 26401.985,E2 26401.985} C_VEL
LIN {X 0,Y 579.921,Z 528.99,A -85,B 0,C 180,E1 26400.587,E2 26400.587} C_VEL
LIN {X 0,Y 576.179,Z 625.533,A -85,B 0,C 180,E1 26398.859,E2 26398.859} C_VEL
LIN {X 0,Y 575.409,Z 647.412,A -85,B 0,C 180,E1 26398.323,E2 26398.323} C_VEL
LIN {X 0,Y 574.297,Z 669.63,A -85,B 0,C 180,E1 26397.589,E2 26397.589} C_VEL
LIN {X 0,Y 573.012,Z 690.725,A -85,B 0,C 180,E1 26396.692,E2 26396.692} C_VEL
LIN {X 0,Y 571.579,Z 710.623,A -85,B 0,C 180,E1 26395.656,E2 26395.656} C_VEL
LIN {X 0,Y 569.998,Z 730.666,A -85,B 0,C 180,E1 26394.401,E2 26394.401} C_VEL
LIN {X 0,Y 568.423,Z 748.96,A -85,B 0,C 180,E1 26393.041,E2 26393.041} C_VEL
LIN {X 0,Y 566.939,Z 765.82,A -85,B 0,C 180,E1 26391.575,E2 26391.575} C_VEL
LIN {X 0,Y 565.41,Z 782.698,A -85,B 0,C 180,E1 26389.849,E2 26389.849} C_VEL
LIN {X 0,Y 564.093,Z 797.426,A -85,B 0,C 180,E1 26388.071,E2 26388.071} C_VEL
LIN {X 0,Y 563.035,Z 810.018,A -85,B 0,C 180,E1 26386.296,E2 26386.296} C_VEL
LIN {X 0,Y 562.119,Z 821.97,A -85,B 0,C 180,E1 26384.315,E2 26384.315} C_VEL
LIN {X 0,Y 561.447,Z 831.988,A -85,B 0,C 180,E1 26382.34,E2 26382.34} C_VEL
LIN {X 0,Y 560.944,Z 840.537,A -85,B 0,C 180,E1 26380.268,E2 26380.268} C_VEL
LIN {X 0,Y 560.624,Z 847.453,A -85,B 0,C 180,E1 26378.164,E2 26378.164} C_VEL
LIN {X 0,Y 560.454,Z 852.782,A -85,B 0,C 180,E1 26376.042,E2 26376.042} C_VEL
LIN {X 0,Y 560.369,Z 856.537,A -85,B 0,C 180,E1 26373.888,E2 26373.888} C_VEL
LIN {X 0,Y 560.329,Z 858.601,A -85,B 0,C 180,E1 26371.738,E2 26371.738} C_VEL
LIN {X 0,Y 560.312,Z 859.114,A -85,B 0,C 180,E1 26369.489,E2 26369.489} C_VEL
LIN {X 0,Y 560.337,Z 858.029,A -85,B 0,C 180,E1 26367.341,E2 26367.341} C_VEL
LIN {X 0,Y 560.397,Z 855.253,A -85,B 0,C 180,E1 26365.19,E2 26365.19} C_VEL
LIN {X 0,Y 560.497,Z 850.869,A -85,B 0,C 180,E1 26363.032,E2 26363.032} C_VEL
LIN {X 0,Y 560.721,Z 845.146,A -85,B 0,C 180,E1 26360.972,E2 26360.972} C_VEL
LIN {X 0,Y 561.142,Z 837.294,A -85,B 0,C 180,E1 26358.801,E2 26358.801} C_VEL
LIN {X 0,Y 561.66,Z 828.399,A -85,B 0,C 180,E1 26356.828,E2 26356.828} C_VEL
LIN {X 0,Y 562.475,Z 817.104,A -85,B 0,C 180,E1 26354.746,E2 26354.746} C_VEL
LIN {X 0,Y 563.456,Z 804.985,A -85,B 0,C 180,E1 26352.868,E2 26352.868} C_VEL
LIN {X 0,Y 564.689,Z 790.849,A -85,B 0,C 180,E1 26351.006,E2 26351.006} C_VEL
LIN {X 0,Y 566.137,Z 774.706,A -85,B 0,C 180,E1 26349.207,E2 26349.207} C_VEL
LIN {X 0,Y 567.626,Z 758.103,A -85,B 0,C 180,E1 26347.636,E2 26347.636} C_VEL
LIN {X 0,Y 569.15,Z 740.648,A -85,B 0,C 180,E1 26346.222,E2 26346.222} C_VEL
LIN {X 0,Y 570.738,Z 721.654,A -85,B 0,C 180,E1 26344.915,E2 26344.915} C_VEL
LIN {X 0,Y 572.175,Z 702.773,A -85,B 0,C 180,E1 26343.816,E2 26343.816} C_VEL
LIN {X 0,Y 573.627,Z 681.462,A -85,B 0,C 180,E1 26342.795,E2 26342.795} C_VEL
LIN {X 0,Y 574.813,Z 660.27,A -85,B 0,C 180,E1 26341.987,E2 26341.987} C_VEL
LIN {X 0,Y 575.742,Z 638.56,A -85,B 0,C 180,E1 26341.348,E2 26341.348} C_VEL
LIN {X 0,Y 576.652,Z 611.573,A -85,B 0,C 180,E1 26340.78,E2 26340.78} C_VEL
LIN {X 0,Y 580.684,Z 509.281,A -85,B 0,C 180,E1 26338.992,E2 26338.992} C_VEL
LIN {X 0,Y 583.434,Z 425.67,A -85,B 0,C 180,E1 26337.696,E2 26337.696} C_VEL
LIN {X 0,Y 585.388,Z 345.041,A -85,B 0,C 180,E1 26336.574,E2 26336.574} C_VEL
LIN {X 0,Y 586.453,Z 339.732,A -85,B 0,C 180,E1 26336.35,E2 26336.35} C_VEL
LIN {X 0,Y 586.414,Z 308.226,A -85,B 0,C 180,E1 26334.255,E2 26334.255} C_VEL
LIN {X 0,Y 587.241,Z 275.669,A -85,B 0,C 180,E1 26331.917,E2 26331.917} C_VEL
LIN {X 0,Y 578.615,Z 253.002,A -85,B 0,C 180,E1 26329.477,E2 26329.477} C_VEL
LIN {X 0,Y 570.838,Z 235.075,A -85,B 0,C 180,E1 26327.513,E2 26327.513} C_VEL
LIN {X 0,Y 562.953,Z 219.066,A -85,B 0,C 180,E1 26325.708,E2 26325.708} C_VEL
LIN {X 0,Y 561.477,Z 215.608,A -85,B 0,C 180,E1 26325.345,E2 26325.345} C_VEL
LIN {X 0,Y 561.429,Z 215.301,A -85,B 0,C 180,E1 26325.285,E2 26325.285} C_VEL
LIN {X 0,Y 561.439,Z 215.303,A -85,B 0,C 180,E1 26322.039,E2 26322.039} C_VEL
LIN {X 0,Y 561.422,Z 215.3,A -85,B 0,C 180,E1 26318.732,E2 26318.732} C_VEL
LIN {X 0,Y 561.438,Z 215.294,A -85,B 0,C 180,E1 26315.346,E2 26315.346} C_VEL
LIN {X 0,Y 561.435,Z 215.283,A -85,B 0,C 180,E1 26312.034,E2 26312.034} C_VEL
LIN {X 0,Y 561.425,Z 215.277,A -85,B 0,C 180,E1 26308.742,E2 26308.742} C_VEL
LIN {X 0,Y 561.438,Z 215.29,A -85,B 0,C 180,E1 26305.417,E2 26305.417} C_VEL
LIN {X 0,Y 561.437,Z 215.282,A -85,B 0,C 180,E1 26302.073,E2 26302.073} C_VEL
LIN {X 0,Y 561.428,Z 215.272,A -85,B 0,C 180,E1 26298.698,E2 26298.698} C_VEL
LIN {X 0,Y 561.433,Z 215.291,A -85,B 0,C 180,E1 26295.389,E2 26295.389} C_VEL
LIN {X 0,Y 561.428,Z 215.266,A -85,B 0,C 180,E1 26292.027,E2 26292.027} C_VEL
LIN {X 0,Y 561.435,Z 215.294,A -85,B 0,C 180,E1 26288.707,E2 26288.707} C_VEL
LIN {X 0,Y 561.418,Z 215.268,A -85,B 0,C 180,E1 26285.519,E2 26285.519} C_VEL
LIN {X 0,Y 561.435,Z 215.295,A -85,B 0,C 180,E1 26282.143,E2 26282.143} C_VEL
LIN {X 0,Y 561.438,Z 215.263,A -85,B 0,C 180,E1 26278.775,E2 26278.775} C_VEL
LIN {X 0,Y 561.415,Z 215.293,A -85,B 0,C 180,E1 26275.505,E2 26275.505} C_VEL
LIN {X 0,Y 561.434,Z 215.265,A -85,B 0,C 180,E1 26272.118,E2 26272.118} C_VEL
LIN {X 0,Y 561.439,Z 215.293,A -85,B 0,C 180,E1 26268.806,E2 26268.806} C_VEL
LIN {X 0,Y 561.411,Z 215.294,A -85,B 0,C 180,E1 26265.561,E2 26265.561} C_VEL
LIN {X 0,Y 561.441,Z 215.295,A -85,B 0,C 180,E1 26262.269,E2 26262.269} C_VEL
LIN {X 0,Y 561.428,Z 215.292,A -85,B 0,C 180,E1 26258.915,E2 26258.915} C_VEL
LIN {X 0,Y 561.406,Z 215.294,A -85,B 0,C 180,E1 26255.594,E2 26255.594} C_VEL
LIN {X 0,Y 561.447,Z 215.292,A -85,B 0,C 180,E1 26252.266,E2 26252.266} C_VEL
LIN {X 0,Y 561.411,Z 215.298,A -85,B 0,C 180,E1 26249.021,E2 26249.021} C_VEL
LIN {X 0,Y 561.404,Z 215.296,A -85,B 0,C 180,E1 26245.626,E2 26245.626} C_VEL
LIN {X 0,Y 561.462,Z 215.418,A -85,B 0,C 180,E1 26242.368,E2 26242.368} C_VEL
LIN {X 0,Y 562.826,Z 218.91,A -85,B 0,C 180,E1 26241.941,E2 26241.941} C_VEL
LIN {X 0,Y 563.963,Z 221.123,A -85,B 0,C 180,E1 26241.644,E2 26241.644} C_VEL
LIN {X 0,Y 570.911,Z 234.738,A -85,B 0,C 180,E1 26239.871,E2 26239.871} C_VEL
LIN {X 0,Y 580.547,Z 253.699,A -85,B 0,C 180,E1 26237.534,E2 26237.534} C_VEL
LIN {X 0,Y 592.791,Z 278.925,A -85,B 0,C 180,E1 26234.698,E2 26234.698} C_VEL
LIN {X 0,Y 594.513,Z 283.316,A -85,B 0,C 180,E1 26234.265,E2 26234.265} C_VEL
LIN {X 0,Y 592.128,Z 310.199,A -85,B 0,C 180,E1 26232.749,E2 26232.749} C_VEL
LIN {X 0,Y 594.916,Z 334.019,A -85,B 0,C 180,E1 26232.149,E2 26232.149} C_VEL
LIN {X 0,Y 588.562,Z 580.572,A -85,B 0,C 180,E1 26228.652,E2 26228.652} C_VEL
LIN {X 0,Y 586.04,Z 692.74,A -85,B 0,C 180,E1 26227.097,E2 26227.097} C_VEL
LIN {X 0,Y 584.879,Z 717.274,A -85,B 0,C 180,E1 26226.591,E2 26226.591} C_VEL
LIN {X 0,Y 583.511,Z 739.8,A -85,B 0,C 180,E1 26225.975,E2 26225.975} C_VEL
LIN {X 0,Y 581.762,Z 763.298,A -85,B 0,C 180,E1 26225.154,E2 26225.154} C_VEL
LIN {X 0,Y 579.948,Z 784.469,A -85,B 0,C 180,E1 26224.258,E2 26224.258} C_VEL
LIN {X 0,Y 577.776,Z 807.376,A -85,B 0,C 180,E1 26223.093,E2 26223.093} C_VEL
LIN {X 0,Y 575.695,Z 827.837,A -85,B 0,C 180,E1 26221.87,E2 26221.87} C_VEL
LIN {X 0,Y 573.372,Z 849.27,A -85,B 0,C 180,E1 26220.379,E2 26220.379} C_VEL
LIN {X 0,Y 571.381,Z 867.088,A -85,B 0,C 180,E1 26218.957,E2 26218.957} C_VEL
LIN {X 0,Y 569.065,Z 887.627,A -85,B 0,C 180,E1 26217.07,E2 26217.07} C_VEL
LIN {X 0,Y 567.25,Z 903.878,A -85,B 0,C 180,E1 26215.362,E2 26215.362} C_VEL
LIN {X 0,Y 565.359,Z 921.592,A -85,B 0,C 180,E1 26213.228,E2 26213.228} C_VEL
LIN {X 0,Y 563.946,Z 935.489,A -85,B 0,C 180,E1 26211.313,E2 26211.313} C_VEL
LIN {X 0,Y 562.613,Z 950.16,A -85,B 0,C 180,E1 26208.98,E2 26208.98} C_VEL
LIN {X 0,Y 561.737,Z 961.076,A -85,B 0,C 180,E1 26206.973,E2 26206.973} C_VEL
LIN {X 0,Y 560.971,Z 972.316,A -85,B 0,C 180,E1 26204.556,E2 26204.556} C_VEL
LIN {X 0,Y 560.518,Z 980.454,A -85,B 0,C 180,E1 26202.465,E2 26202.465} C_VEL
LIN {X 0,Y 560.186,Z 988.207,A -85,B 0,C 180,E1 26200.074,E2 26200.074} C_VEL
LIN {X 0,Y 559.997,Z 993.849,A -85,B 0,C 180,E1 26197.799,E2 26197.799} C_VEL
LIN {X 0,Y 559.936,Z 997.751,A -85,B 0,C 180,E1 26195.739,E2 26195.739} C_VEL
LIN {X 0,Y 559.901,Z 1000.905,A -85,B 0,C 180,E1 26193.276,E2 26193.276} C_VEL
LIN {X 0,Y 559.899,Z 1002.184,A -85,B 0,C 180,E1 26191.023,E2 26191.023} C_VEL
LIN {X 0,Y 559.894,Z 1002.207,A -85,B 0,C 180,E1 26189.079,E2 26189.079} C_VEL
LIN {X 0,Y 559.891,Z 1001.05,A -85,B 0,C 180,E1 26186.929,E2 26186.929} C_VEL
LIN {X 0,Y 559.921,Z 998.071,A -85,B 0,C 180,E1 26184.466,E2 26184.466} C_VEL
LIN {X 0,Y 559.985,Z 994.242,A -85,B 0,C 180,E1 26182.407,E2 26182.407} C_VEL
LIN {X 0,Y 560.164,Z 989.198,A -85,B 0,C 180,E1 26180.341,E2 26180.341} C_VEL
LIN {X 0,Y 560.469,Z 981.347,A -85,B 0,C 180,E1 26177.847,E2 26177.847} C_VEL
LIN {X 0,Y 560.892,Z 973.239,A -85,B 0,C 180,E1 26175.758,E2 26175.758} C_VEL
LIN {X 0,Y 561.577,Z 962.61,A -85,B 0,C 180,E1 26173.448,E2 26173.448} C_VEL
LIN {X 0,Y 562.482,Z 950.414,A -85,B 0,C 180,E1 26171.231,E2 26171.231} C_VEL
LIN {X 0,Y 563.614,Z 936.977,A -85,B 0,C 180,E1 26169.109,E2 26169.109} C_VEL
LIN {X 0,Y 564.998,Z 922.006,A -85,B 0,C 180,E1 26167.087,E2 26167.087} C_VEL
LIN {X 0,Y 566.588,Z 905.371,A -85,B 0,C 180,E1 26165.106,E2 26165.106} C_VEL
LIN {X 0,Y 568.331,Z 887.591,A -85,B 0,C 180,E1 26163.287,E2 26163.287} C_VEL
LIN {X 0,Y 570.202,Z 868.597,A -85,B 0,C 180,E1 26161.569,E2 26161.569} C_VEL
LIN {X 0,Y 572.135,Z 848.552,A -85,B 0,C 180,E1 26160.011,E2 26160.011} C_VEL
LIN {X 0,Y 574.143,Z 827.442,A -85,B 0,C 180,E1 26158.579,E2 26158.579} C_VEL
LIN {X 0,Y 575.917,Z 806.696,A -85,B 0,C 180,E1 26157.373,E2 26157.373} C_VEL
LIN {X 0,Y 577.801,Z 783.543,A -85,B 0,C 180,E1 26156.222,E2 26156.222} C_VEL
LIN {X 0,Y 579.366,Z 761.816,A -85,B 0,C 180,E1 26155.33,E2 26155.33} C_VEL
LIN {X 0,Y 580.894,Z 737.628,A -85,B 0,C 180,E1 26154.513,E2 26154.513} C_VEL
LIN {X 0,Y 582,Z 715.071,A -85,B 0,C 180,E1 26153.924,E2 26153.924} C_VEL
LIN {X 0,Y 582.938,Z 690.138,A -85,B 0,C 180,E1 26153.441,E2 26153.441} C_VEL
LIN {X 0,Y 585.653,Z 533.304,A -85,B 0,C 180,E1 26151.348,E2 26151.348} C_VEL
LIN {X 0,Y 588.603,Z 421.987,A -85,B 0,C 180,E1 26149.699,E2 26149.699} C_VEL
LIN {X 0,Y 592.073,Z 331.436,A -85,B 0,C 180,E1 26148.223,E2 26148.223} C_VEL
LIN {X 0,Y 592.101,Z 329.405,A -85,B 0,C 180,E1 26148.136,E2 26148.136} C_VEL
LIN {X 0,Y 597.294,Z 307.596,A -85,B 0,C 180,E1 26146.526,E2 26146.526} C_VEL
LIN {X 0,Y 602.859,Z 290.39,A -85,B 0,C 180,E1 26145.137,E2 26145.137} C_VEL
LIN {X 0,Y 601.971,Z 285.99,A -85,B 0,C 180,E1 26143.972,E2 26143.972} C_VEL
LIN {X 0,Y 601.511,Z 283.922,A -85,B 0,C 180,E1 26143.095,E2 26143.095} C_VEL
LIN {X 0,Y 601.513,Z 282.186,A -85,B 0,C 180,E1 26141.804,E2 26141.804} C_VEL
LIN {X 0,Y 601.236,Z 284.033,A -85,B 0,C 180,E1 26140.311,E2 26140.311} C_VEL
LIN {X 0,Y 601.422,Z 287.216,A -85,B 0,C 180,E1 26139.181,E2 26139.181} C_VEL
LIN {X 0,Y 601.421,Z 288.711,A -85,B 0,C 180,E1 26138.813,E2 26138.813} C_VEL
LIN {X 0,Y 594.149,Z 309.834,A -85,B 0,C 180,E1 26136.806,E2 26136.806} C_VEL
LIN {X 0,Y 587.473,Z 337.328,A -85,B 0,C 180,E1 26134.407,E2 26134.407} C_VEL
LIN {X 0,Y 581.912,Z 370.482,A -85,B 0,C 180,E1 26131.722,E2 26131.722} C_VEL
LIN {X 0,Y 576.869,Z 412.068,A -85,B 0,C 180,E1 26128.581,E2 26128.581} C_VEL
LIN {X 0,Y 576.6,Z 416.359,A -85,B 0,C 180,E1 26128.297,E2 26128.297} C_VEL
LIN {X 0,Y 579.297,Z 444.577,A -85,B 0,C 180,E1 26127.133,E2 26127.133} C_VEL
LIN {X 0,Y 581.891,Z 479.086,A -85,B 0,C 180,E1 26125.899,E2 26125.899} C_VEL
LIN {X 0,Y 582.738,Z 496.873,A -85,B 0,C 180,E1 26125.351,E2 26125.351} C_VEL
LIN {X 0,Y 575.952,Z 603.696,A -85,B 0,C 180,E1 26123.162,E2 26123.162} C_VEL
LIN {X 0,Y 571.963,Z 688.572,A -85,B 0,C 180,E1 26121.474,E2 26121.474} C_VEL
LIN {X 0,Y 570.83,Z 711.243,A -85,B 0,C 180,E1 26120.824,E2 26120.824} C_VEL
LIN {X 0,Y 569.701,Z 732.552,A -85,B 0,C 180,E1 26120.014,E2 26120.014} C_VEL
LIN {X 0,Y 568.545,Z 752.867,A -85,B 0,C 180,E1 26119.041,E2 26119.041} C_VEL
LIN {X 0,Y 567.462,Z 771.005,A -85,B 0,C 180,E1 26117.96,E2 26117.96} C_VEL
LIN {X 0,Y 566.378,Z 788.148,A -85,B 0,C 180,E1 26116.724,E2 26116.724} C_VEL
LIN {X 0,Y 565.418,Z 802.733,A -85,B 0,C 180,E1 26115.467,E2 26115.467} C_VEL
LIN {X 0,Y 564.477,Z 816.474,A -85,B 0,C 180,E1 26114.045,E2 26114.045} C_VEL
LIN {X 0,Y 563.63,Z 828.893,A -85,B 0,C 180,E1 26112.5,E2 26112.5} C_VEL
LIN {X 0,Y 562.93,Z 839.125,A -85,B 0,C 180,E1 26110.956,E2 26110.956} C_VEL
LIN {X 0,Y 562.29,Z 848.446,A -85,B 0,C 180,E1 26109.209,E2 26109.209} C_VEL
LIN {X 0,Y 561.818,Z 855.758,A -85,B 0,C 180,E1 26107.465,E2 26107.465} C_VEL
LIN {X 0,Y 561.465,Z 861.497,A -85,B 0,C 180,E1 26105.621,E2 26105.621} C_VEL
LIN {X 0,Y 561.197,Z 865.371,A -85,B 0,C 180,E1 26103.78,E2 26103.78} C_VEL
LIN {X 0,Y 561.012,Z 867.549,A -85,B 0,C 180,E1 26101.838,E2 26101.838} C_VEL
LIN {X 0,Y 560.919,Z 867.885,A -85,B 0,C 180,E1 26100,E2 26100} C_VEL
LIN {X 0,Y 560.867,Z 866.419,A -85,B 0,C 180,E1 26098.059,E2 26098.059} C_VEL
LIN {X 0,Y 560.893,Z 863.09,A -85,B 0,C 180,E1 26096.116,E2 26096.116} C_VEL
LIN {X 0,Y 561.01,Z 858.171,A -85,B 0,C 180,E1 26094.272,E2 26094.272} C_VEL
LIN {X 0,Y 561.215,Z 851.408,A -85,B 0,C 180,E1 26092.424,E2 26092.424} C_VEL
LIN {X 0,Y 561.545,Z 843.168,A -85,B 0,C 180,E1 26090.675,E2 26090.675} C_VEL
LIN {X 0,Y 562.042,Z 832.882,A -85,B 0,C 180,E1 26088.923,E2 26088.923} C_VEL
LIN {X 0,Y 562.681,Z 821.036,A -85,B 0,C 180,E1 26087.27,E2 26087.27} C_VEL
LIN {X 0,Y 563.459,Z 807.62,A -85,B 0,C 180,E1 26085.72,E2 26085.72} C_VEL
LIN {X 0,Y 564.359,Z 792.576,A -85,B 0,C 180,E1 26084.272,E2 26084.272} C_VEL
LIN {X 0,Y 565.367,Z 775.732,A -85,B 0,C 180,E1 26082.927,E2 26082.927} C_VEL
LIN {X 0,Y 566.359,Z 758.188,A -85,B 0,C 180,E1 26081.773,E2 26081.773} C_VEL
LIN {X 0,Y 567.343,Z 740.261,A -85,B 0,C 180,E1 26080.811,E2 26080.811} C_VEL
LIN {X 0,Y 568.303,Z 720.779,A -85,B 0,C 180,E1 26079.974,E2 26079.974} C_VEL
LIN {X 0,Y 569.15,Z 700.322,A -85,B 0,C 180,E1 26079.307,E2 26079.307} C_VEL
LIN {X 0,Y 569.857,Z 679.643,A -85,B 0,C 180,E1 26078.834,E2 26078.834} C_VEL
LIN {X 0,Y 574.449,Z 491.167,A -85,B 0,C 180,E1 26075.896,E2 26075.896} C_VEL
LIN {X 0,Y 570.367,Z 454.133,A -85,B 0,C 180,E1 26075.063,E2 26075.063} C_VEL
LIN {X 0,Y 573.177,Z 401.497,A -85,B 0,C 180,E1 26071.616,E2 26071.616} C_VEL
LIN {X 0,Y 576.239,Z 350.111,A -85,B 0,C 180,E1 26068.21,E2 26068.21} C_VEL
LIN {X 0,Y 579.604,Z 298.699,A -85,B 0,C 180,E1 26064.756,E2 26064.756} C_VEL
LIN {X 0,Y 581.653,Z 266.917,A -85,B 0,C 180,E1 26062.58,E2 26062.58} C_VEL
LIN {X 0,Y 573.104,Z 244.424,A -85,B 0,C 180,E1 26060.301,E2 26060.301} C_VEL
LIN {X 0,Y 564.311,Z 222.551,A -85,B 0,C 180,E1 26057.938,E2 26057.938} C_VEL
LIN {X 0,Y 563.532,Z 221.076,A -85,B 0,C 180,E1 26057.76,E2 26057.76} C_VEL
LIN {X 0,Y 561.352,Z 218.415,A -85,B 0,C 180,E1 26057.345,E2 26057.345} C_VEL
LIN {X 0,Y 557.652,Z 216.768,A -85,B 0,C 180,E1 26056.765,E2 26056.765} C_VEL
LIN {X 0,Y 554.482,Z 216.314,A -85,B 0,C 180,E1 26056.124,E2 26056.124} C_VEL
LIN {X 0,Y 553.485,Z 216.285,A -85,B 0,C 180,E1 26055.578,E2 26055.578} C_VEL
LIN {X 0,Y 553.521,Z 216.448,A -85,B 0,C 180,E1 26055.276,E2 26055.276} C_VEL
LIN {X 0,Y 554.89,Z 219.882,A -85,B 0,C 180,E1 26054.913,E2 26054.913} C_VEL
LIN {X 0,Y 555.954,Z 221.762,A -85,B 0,C 180,E1 26054.686,E2 26054.686} C_VEL
LIN {X 0,Y 563.877,Z 237.896,A -85,B 0,C 180,E1 26052.841,E2 26052.841} C_VEL
LIN {X 0,Y 571.245,Z 254.839,A -85,B 0,C 180,E1 26050.949,E2 26050.949} C_VEL
LIN {X 0,Y 579.569,Z 276.454,A -85,B 0,C 180,E1 26048.599,E2 26048.599} C_VEL
LIN {X 0,Y 580.664,Z 279.683,A -85,B 0,C 180,E1 26048.258,E2 26048.258} C_VEL
LIN {X 0,Y 579.819,Z 321.696,A -85,B 0,C 180,E1 26045.289,E2 26045.289} C_VEL
LIN {X 0,Y 579.92,Z 342.208,A -85,B 0,C 180,E1 26043.962,E2 26043.962} C_VEL
LIN {X 0,Y 578.554,Z 349.119,A -85,B 0,C 180,E1 26043.708,E2 26043.708} C_VEL
LIN {X 0,Y 576.214,Z 442.69,A -85,B 0,C 180,E1 26042.398,E2 26042.398} C_VEL
LIN {X 0,Y 573.102,Z 528.948,A -85,B 0,C 180,E1 26041.006,E2 26041.006} C_VEL
LIN {X 0,Y 569.13,Z 626.101,A -85,B 0,C 180,E1 26039.233,E2 26039.233} C_VEL
LIN {X 0,Y 568.324,Z 648.408,A -85,B 0,C 180,E1 26038.683,E2 26038.683} C_VEL
LIN {X 0,Y 567.159,Z 670.619,A -85,B 0,C 180,E1 26037.938,E2 26037.938} C_VEL
LIN {X 0,Y 565.851,Z 691.3,A -85,B 0,C 180,E1 26037.051,E2 26037.051} C_VEL
LIN {X 0,Y 564.367,Z 711.189,A -85,B 0,C 180,E1 26036.008,E2 26036.008} C_VEL
LIN {X 0,Y 562.705,Z 731.31,A -85,B 0,C 180,E1 26034.738,E2 26034.738} C_VEL
LIN {X 0,Y 561.058,Z 749.599,A -85,B 0,C 180,E1 26033.367,E2 26033.367} C_VEL
LIN {X 0,Y 559.43,Z 767.104,A -85,B 0,C 180,E1 26031.825,E2 26031.825} C_VEL
LIN {X 0,Y 557.857,Z 783.435,A -85,B 0,C 180,E1 26030.129,E2 26030.129} C_VEL
LIN {X 0,Y 556.535,Z 797.387,A -85,B 0,C 180,E1 26028.434,E2 26028.434} C_VEL
LIN {X 0,Y 555.334,Z 810.837,A -85,B 0,C 180,E1 26026.528,E2 26026.528} C_VEL
LIN {X 0,Y 554.391,Z 822.259,A -85,B 0,C 180,E1 26024.626,E2 26024.626} C_VEL
LIN {X 0,Y 553.621,Z 832.861,A -85,B 0,C 180,E1 26022.517,E2 26022.517} C_VEL
LIN {X 0,Y 553.078,Z 841.431,A -85,B 0,C 180,E1 26020.416,E2 26020.416} C_VEL
LIN {X 0,Y 552.731,Z 848.333,A -85,B 0,C 180,E1 26018.299,E2 26018.299} C_VEL
LIN {X 0,Y 552.538,Z 853.742,A -85,B 0,C 180,E1 26016.129,E2 26016.129} C_VEL
LIN {X 0,Y 552.438,Z 857.514,A -85,B 0,C 180,E1 26013.944,E2 26013.944} C_VEL
LIN {X 0,Y 552.394,Z 859.597,A -85,B 0,C 180,E1 26011.763,E2 26011.763} C_VEL
LIN {X 0,Y 552.374,Z 860.115,A -85,B 0,C 180,E1 26009.481,E2 26009.481} C_VEL
LIN {X 0,Y 552.403,Z 859.016,A -85,B 0,C 180,E1 26007.303,E2 26007.303} C_VEL
LIN {X 0,Y 552.47,Z 856.226,A -85,B 0,C 180,E1 26005.12,E2 26005.12} C_VEL
LIN {X 0,Y 552.584,Z 851.812,A -85,B 0,C 180,E1 26002.932,E2 26002.932} C_VEL
LIN {X 0,Y 552.848,Z 845.705,A -85,B 0,C 180,E1 26000.737,E2 26000.737} C_VEL
LIN {X 0,Y 553.292,Z 838.188,A -85,B 0,C 180,E1 25998.64,E2 25998.64} C_VEL
LIN {X 0,Y 553.898,Z 828.756,A -85,B 0,C 180,E1 25996.534,E2 25996.534} C_VEL
LIN {X 0,Y 554.737,Z 817.93,A -85,B 0,C 180,E1 25994.528,E2 25994.528} C_VEL
LIN {X 0,Y 555.845,Z 805.023,A -85,B 0,C 180,E1 25992.518,E2 25992.518} C_VEL
LIN {X 0,Y 557.108,Z 791.427,A -85,B 0,C 180,E1 25990.717,E2 25990.717} C_VEL
LIN {X 0,Y 558.588,Z 775.957,A -85,B 0,C 180,E1 25988.967,E2 25988.967} C_VEL
LIN {X 0,Y 560.214,Z 758.821,A -85,B 0,C 180,E1 25987.324,E2 25987.324} C_VEL
LIN {X 0,Y 561.811,Z 741.377,A -85,B 0,C 180,E1 25985.898,E2 25985.898} C_VEL
LIN {X 0,Y 563.487,Z 722.246,A -85,B 0,C 180,E1 25984.569,E2 25984.569} C_VEL
LIN {X 0,Y 565.053,Z 702.232,A -85,B 0,C 180,E1 25983.404,E2 25983.404} C_VEL
LIN {X 0,Y 566.461,Z 682.502,A -85,B 0,C 180,E1 25982.453,E2 25982.453} C_VEL
LIN {X 0,Y 567.706,Z 661.32,A -85,B 0,C 180,E1 25981.634,E2 25981.634} C_VEL
LIN {X 0,Y 568.667,Z 639.573,A -85,B 0,C 180,E1 25980.986,E2 25980.986} C_VEL
LIN {X 0,Y 569.618,Z 612.327,A -85,B 0,C 180,E1 25980.405,E2 25980.405} C_VEL
LIN {X 0,Y 573.742,Z 513.351,A -85,B 0,C 180,E1 25978.637,E2 25978.637} C_VEL
LIN {X 0,Y 576.592,Z 431.128,A -85,B 0,C 180,E1 25977.339,E2 25977.339} C_VEL
LIN {X 0,Y 578.708,Z 347.779,A -85,B 0,C 180,E1 25976.166,E2 25976.166} C_VEL
LIN {X 0,Y 580.002,Z 341.168,A -85,B 0,C 180,E1 25975.884,E2 25975.884} C_VEL
LIN {X 0,Y 579.996,Z 308.239,A -85,B 0,C 180,E1 25973.688,E2 25973.688} C_VEL
LIN {X 0,Y 580.613,Z 279.112,A -85,B 0,C 180,E1 25971.589,E2 25971.589} C_VEL
LIN {X 0,Y 572.14,Z 256.868,A -85,B 0,C 180,E1 25969.177,E2 25969.177} C_VEL
LIN {X 0,Y 564.396,Z 238.99,A -85,B 0,C 180,E1 25967.176,E2 25967.176} C_VEL
LIN {X 0,Y 557.007,Z 223.955,A -85,B 0,C 180,E1 25965.452,E2 25965.452} C_VEL
LIN {X 0,Y 555.267,Z 220.416,A -85,B 0,C 180,E1 25965.048,E2 25965.048} C_VEL
LIN {X 0,Y 553.664,Z 217.25,A -85,B 0,C 180,E1 25964.684,E2 25964.684} C_VEL
LIN {X 0,Y 553.487,Z 216.285,A -85,B 0,C 180,E1 25964.581,E2 25964.581} C_VEL
LIN {X 0,Y 553.485,Z 216.28,A -85,B 0,C 180,E1 25961.116,E2 25961.116} C_VEL
LIN {X 0,Y 553.497,Z 216.278,A -85,B 0,C 180,E1 25957.867,E2 25957.867} C_VEL
LIN {X 0,Y 553.49,Z 216.287,A -85,B 0,C 180,E1 25954.536,E2 25954.536} C_VEL
LIN {X 0,Y 553.494,Z 216.282,A -85,B 0,C 180,E1 25951.098,E2 25951.098} C_VEL
LIN {X 0,Y 553.491,Z 216.267,A -85,B 0,C 180,E1 25947.78,E2 25947.78} C_VEL
LIN {X 0,Y 553.496,Z 216.264,A -85,B 0,C 180,E1 25944.429,E2 25944.429} C_VEL
LIN {X 0,Y 553.495,Z 216.28,A -85,B 0,C 180,E1 25940.958,E2 25940.958} C_VEL
LIN {X 0,Y 553.486,Z 216.257,A -85,B 0,C 180,E1 25937.668,E2 25937.668} C_VEL
LIN {X 0,Y 553.502,Z 216.277,A -85,B 0,C 180,E1 25934.329,E2 25934.329} C_VEL
LIN {X 0,Y 553.496,Z 216.265,A -85,B 0,C 180,E1 25930.934,E2 25930.934} C_VEL
LIN {X 0,Y 553.48,Z 216.271,A -85,B 0,C 180,E1 25927.578,E2 25927.578} C_VEL
LIN {X 0,Y 553.495,Z 216.269,A -85,B 0,C 180,E1 25924.248,E2 25924.248} C_VEL
LIN {X 0,Y 553.5,Z 216.268,A -85,B 0,C 180,E1 25920.828,E2 25920.828} C_VEL
LIN {X 0,Y 553.478,Z 216.281,A -85,B 0,C 180,E1 25917.472,E2 25917.472} C_VEL
LIN {X 0,Y 553.494,Z 216.261,A -85,B 0,C 180,E1 25914.09,E2 25914.09} C_VEL
LIN {X 0,Y 553.502,Z 216.274,A -85,B 0,C 180,E1 25910.748,E2 25910.748} C_VEL
LIN {X 0,Y 553.471,Z 216.285,A -85,B 0,C 180,E1 25907.479,E2 25907.479} C_VEL
LIN {X 0,Y 553.501,Z 216.278,A -85,B 0,C 180,E1 25904.17,E2 25904.17} C_VEL
LIN {X 0,Y 553.497,Z 216.278,A -85,B 0,C 180,E1 25900.805,E2 25900.805} C_VEL
LIN {X 0,Y 553.467,Z 216.289,A -85,B 0,C 180,E1 25897.48,E2 25897.48} C_VEL
LIN {X 0,Y 553.499,Z 216.285,A -85,B 0,C 180,E1 25894.11,E2 25894.11} C_VEL
LIN {X 0,Y 553.497,Z 216.278,A -85,B 0,C 180,E1 25890.755,E2 25890.755} C_VEL
LIN {X 0,Y 553.46,Z 216.291,A -85,B 0,C 180,E1 25887.427,E2 25887.427} C_VEL
LIN {X 0,Y 553.501,Z 216.277,A -85,B 0,C 180,E1 25884.176,E2 25884.176} C_VEL
LIN {X 0,Y 553.476,Z 216.421,A -85,B 0,C 180,E1 25883.184,E2 25883.184} C_VEL
LIN {X 0,Y 554.881,Z 219.897,A -85,B 0,C 180,E1 25882.737,E2 25882.737} C_VEL
LIN {X 0,Y 556.036,Z 221.965,A -85,B 0,C 180,E1 25882.439,E2 25882.439} C_VEL
LIN {X 0,Y 565.205,Z 240.074,A -85,B 0,C 180,E1 25880.046,E2 25880.046} C_VEL
LIN {X 0,Y 575.598,Z 260.783,A -85,B 0,C 180,E1 25877.488,E2 25877.488} C_VEL
LIN {X 0,Y 586.882,Z 284.08,A -85,B 0,C 180,E1 25874.857,E2 25874.857} C_VEL
LIN {X 0,Y 587.893,Z 286.655,A -85,B 0,C 180,E1 25874.599,E2 25874.599} C_VEL
LIN {X 0,Y 585.671,Z 310.899,A -85,B 0,C 180,E1 25873.222,E2 25873.222} C_VEL
LIN {X 0,Y 588.469,Z 335.301,A -85,B 0,C 180,E1 25872.597,E2 25872.597} C_VEL
LIN {X 0,Y 581.957,Z 573.346,A -85,B 0,C 180,E1 25869.171,E2 25869.171} C_VEL
LIN {X 0,Y 579.108,Z 692.876,A -85,B 0,C 180,E1 25867.49,E2 25867.49} C_VEL
LIN {X 0,Y 577.898,Z 717.248,A -85,B 0,C 180,E1 25866.981,E2 25866.981} C_VEL
LIN {X 0,Y 576.472,Z 739.786,A -85,B 0,C 180,E1 25866.357,E2 25866.357} C_VEL
LIN {X 0,Y 574.658,Z 763.111,A -85,B 0,C 180,E1 25865.532,E2 25865.532} C_VEL
LIN {X 0,Y 572.77,Z 784.233,A -85,B 0,C 180,E1 25864.627,E2 25864.627} C_VEL
LIN {X 0,Y 570.474,Z 807.48,A -85,B 0,C 180,E1 25863.431,E2 25863.431} C_VEL
LIN {X 0,Y 568.337,Z 827.671,A -85,B 0,C 180,E1 25862.213,E2 25862.213} C_VEL
LIN {X 0,Y 565.924,Z 849.068,A -85,B 0,C 180,E1 25860.705,E2 25860.705} C_VEL
LIN {X 0,Y 563.747,Z 867.705,A -85,B 0,C 180,E1 25859.193,E2 25859.193} C_VEL
LIN {X 0,Y 561.419,Z 887.384,A -85,B 0,C 180,E1 25857.355,E2 25857.355} C_VEL
LIN {X 0,Y 559.602,Z 903.013,A -85,B 0,C 180,E1 25855.69,E2 25855.69} C_VEL
LIN {X 0,Y 557.635,Z 920.451,A -85,B 0,C 180,E1 25853.569,E2 25853.569} C_VEL
LIN {X 0,Y 556.167,Z 934.394,A -85,B 0,C 180,E1 25851.626,E2 25851.626} C_VEL
LIN {X 0,Y 554.754,Z 949.139,A -85,B 0,C 180,E1 25849.259,E2 25849.259} C_VEL
LIN {X 0,Y 553.786,Z 960.626,A -85,B 0,C 180,E1 25847.116,E2 25847.116} C_VEL
LIN {X 0,Y 553,Z 971.81,A -85,B 0,C 180,E1 25844.663,E2 25844.663} C_VEL
LIN {X 0,Y 552.537,Z 979.916,A -85,B 0,C 180,E1 25842.542,E2 25842.542} C_VEL
LIN {X 0,Y 552.204,Z 987.598,A -85,B 0,C 180,E1 25840.116,E2 25840.116} C_VEL
LIN {X 0,Y 552.019,Z 993.268,A -85,B 0,C 180,E1 25837.776,E2 25837.776} C_VEL
LIN {X 0,Y 551.967,Z 997.063,A -85,B 0,C 180,E1 25835.718,E2 25835.718} C_VEL
LIN {X 0,Y 551.94,Z 1000.124,A -85,B 0,C 180,E1 25833.219,E2 25833.219} C_VEL
LIN {X 0,Y 551.945,Z 1001.33,A -85,B 0,C 180,E1 25831.038,E2 25831.038} C_VEL
LIN {X 0,Y 551.947,Z 1001.321,A -85,B 0,C 180,E1 25828.962,E2 25828.962} C_VEL
LIN {X 0,Y 551.954,Z 999.888,A -85,B 0,C 180,E1 25826.531,E2 25826.531} C_VEL
LIN {X 0,Y 551.991,Z 996.633,A -85,B 0,C 180,E1 25824.074,E2 25824.074} C_VEL
LIN {X 0,Y 552.066,Z 992.393,A -85,B 0,C 180,E1 25821.878,E2 25821.878} C_VEL
LIN {X 0,Y 552.28,Z 985.766,A -85,B 0,C 180,E1 25819.358,E2 25819.358} C_VEL
LIN {X 0,Y 552.616,Z 978.362,A -85,B 0,C 180,E1 25817.141,E2 25817.141} C_VEL
LIN {X 0,Y 553.181,Z 968.437,A -85,B 0,C 180,E1 25814.698,E2 25814.698} C_VEL
LIN {X 0,Y 553.964,Z 957.45,A -85,B 0,C 180,E1 25812.456,E2 25812.456} C_VEL
LIN {X 0,Y 555.052,Z 943.909,A -85,B 0,C 180,E1 25810.094,E2 25810.094} C_VEL
LIN {X 0,Y 556.223,Z 930.908,A -85,B 0,C 180,E1 25808.154,E2 25808.154} C_VEL
LIN {X 0,Y 557.734,Z 915.298,A -85,B 0,C 180,E1 25806.098,E2 25806.098} C_VEL
LIN {X 0,Y 559.464,Z 898.041,A -85,B 0,C 180,E1 25804.146,E2 25804.146} C_VEL
LIN {X 0,Y 561.395,Z 879.458,A -85,B 0,C 180,E1 25802.299,E2 25802.299} C_VEL
LIN {X 0,Y 563.277,Z 861.157,A -85,B 0,C 180,E1 25800.72,E2 25800.72} C_VEL
LIN {X 0,Y 565.361,Z 840.323,A -85,B 0,C 180,E1 25799.143,E2 25799.143} C_VEL
LIN {X 0,Y 567.275,Z 820.217,A -85,B 0,C 180,E1 25797.838,E2 25797.838} C_VEL
LIN {X 0,Y 569.313,Z 798.034,A -85,B 0,C 180,E1 25796.591,E2 25796.591} C_VEL
LIN {X 0,Y 571.068,Z 776.145,A -85,B 0,C 180,E1 25795.56,E2 25795.56} C_VEL
LIN {X 0,Y 572.778,Z 752.775,A -85,B 0,C 180,E1 25794.641,E2 25794.641} C_VEL
LIN {X 0,Y 574.146,Z 730.177,A -85,B 0,C 180,E1 25793.931,E2 25793.931} C_VEL
LIN {X 0,Y 575.44,Z 704.455,A -85,B 0,C 180,E1 25793.315,E2 25793.315} C_VEL
LIN {X 0,Y 576.164,Z 682.191,A -85,B 0,C 180,E1 25792.938,E2 25792.938} C_VEL
LIN {X 0,Y 578.616,Z 550.242,A -85,B 0,C 180,E1 25791.149,E2 25791.149} C_VEL
LIN {X 0,Y 581.652,Z 443.014,A -85,B 0,C 180,E1 25789.532,E2 25789.532} C_VEL
LIN {X 0,Y 585.823,Z 345.904,A -85,B 0,C 180,E1 25787.926,E2 25787.926} C_VEL
LIN {X 0,Y 586.386,Z 332.55,A -85,B 0,C 180,E1 25787.675,E2 25787.675} C_VEL
LIN {X 0,Y 592.083,Z 311.14,A -85,B 0,C 180,E1 25786.046,E2 25786.046} C_VEL
LIN {X 0,Y 597.7,Z 295.313,A -85,B 0,C 180,E1 25784.719,E2 25784.719} C_VEL
LIN {X 0,Y 597.063,Z 291.289,A -85,B 0,C 180,E1 25783.496,E2 25783.496} C_VEL
LIN {X 0,Y 596.806,Z 289.008,A -85,B 0,C 180,E1 25782.08,E2 25782.08} C_VEL
LIN {X 0,Y 596.743,Z 288.9,A -85,B 0,C 180,E1 25781.642,E2 25781.642} C_VEL
LIN {X 0,Y 596.491,Z 290.948,A -85,B 0,C 180,E1 25780.194,E2 25780.194} C_VEL
LIN {X 0,Y 596.557,Z 293.762,A -85,B 0,C 180,E1 25779.221,E2 25779.221} C_VEL
LIN {X 0,Y 589.076,Z 313.361,A -85,B 0,C 180,E1 25777.299,E2 25777.299} C_VEL
LIN {X 0,Y 582.028,Z 339.205,A -85,B 0,C 180,E1 25774.969,E2 25774.969} C_VEL
LIN {X 0,Y 575.944,Z 371.471,A -85,B 0,C 180,E1 25772.277,E2 25772.277} C_VEL
LIN {X 0,Y 570.647,Z 410.651,A -85,B 0,C 180,E1 25769.238,E2 25769.238} C_VEL
LIN {X 0,Y 570.699,Z 414.084,A -85,B 0,C 180,E1 25769.052,E2 25769.052} C_VEL
LIN {X 0,Y 573.177,Z 442.286,A -85,B 0,C 180,E1 25767.816,E2 25767.816} C_VEL
LIN {X 0,Y 575.473,Z 475.641,A -85,B 0,C 180,E1 25766.562,E2 25766.562} C_VEL
LIN {X 0,Y 576.496,Z 497.783,A -85,B 0,C 180,E1 25765.838,E2 25765.838} C_VEL
LIN {X 0,Y 569.301,Z 603.387,A -85,B 0,C 180,E1 25763.613,E2 25763.613} C_VEL
LIN {X 0,Y 564.916,Z 688.685,A -85,B 0,C 180,E1 25761.858,E2 25761.858} C_VEL
LIN {X 0,Y 563.657,Z 711.807,A -85,B 0,C 180,E1 25761.178,E2 25761.178} C_VEL
LIN {X 0,Y 562.504,Z 732.325,A -85,B 0,C 180,E1 25760.39,E2 25760.39} C_VEL
LIN {X 0,Y 561.315,Z 751.668,A -85,B 0,C 180,E1 25759.458,E2 25759.458} C_VEL
LIN {X 0,Y 560.101,Z 771.034,A -85,B 0,C 180,E1 25758.312,E2 25758.312} C_VEL
LIN {X 0,Y 558.939,Z 788.319,A -85,B 0,C 180,E1 25757.061,E2 25757.061} C_VEL
LIN {X 0,Y 557.837,Z 803.862,A -85,B 0,C 180,E1 25755.704,E2 25755.704} C_VEL
LIN {X 0,Y 556.901,Z 816.943,A -85,B 0,C 180,E1 25754.346,E2 25754.346} C_VEL
LIN {X 0,Y 555.979,Z 829.452,A -85,B 0,C 180,E1 25752.78,E2 25752.78} C_VEL
LIN {X 0,Y 555.17,Z 840.396,A -85,B 0,C 180,E1 25751.111,E2 25751.111} C_VEL
LIN {X 0,Y 554.524,Z 849.241,A -85,B 0,C 180,E1 25749.444,E2 25749.444} C_VEL
LIN {X 0,Y 553.997,Z 856.608,A -85,B 0,C 180,E1 25747.675,E2 25747.675} C_VEL
LIN {X 0,Y 553.605,Z 862.426,A -85,B 0,C 180,E1 25745.805,E2 25745.805} C_VEL
LIN {X 0,Y 553.309,Z 866.365,A -85,B 0,C 180,E1 25743.938,E2 25743.938} C_VEL
LIN {X 0,Y 553.114,Z 868.524,A -85,B 0,C 180,E1 25742.072,E2 25742.072} C_VEL
LIN {X 0,Y 552.996,Z 868.976,A -85,B 0,C 180,E1 25740.207,E2 25740.207} C_VEL
LIN {X 0,Y 552.93,Z 867.747,A -85,B 0,C 180,E1 25738.342,E2 25738.342} C_VEL
LIN {X 0,Y 552.943,Z 864.851,A -85,B 0,C 180,E1 25736.475,E2 25736.475} C_VEL
LIN {X 0,Y 553.04,Z 860.244,A -85,B 0,C 180,E1 25734.605,E2 25734.605} C_VEL
LIN {X 0,Y 553.236,Z 853.821,A -85,B 0,C 180,E1 25732.732,E2 25732.732} C_VEL
LIN {X 0,Y 553.552,Z 845.926,A -85,B 0,C 180,E1 25730.958,E2 25730.958} C_VEL
LIN {X 0,Y 554.037,Z 836.053,A -85,B 0,C 180,E1 25729.182,E2 25729.182} C_VEL
LIN {X 0,Y 554.663,Z 824.668,A -85,B 0,C 180,E1 25727.507,E2 25727.507} C_VEL
LIN {X 0,Y 555.429,Z 811.79,A -85,B 0,C 180,E1 25725.935,E2 25725.935} C_VEL
LIN {X 0,Y 556.34,Z 797.092,A -85,B 0,C 180,E1 25724.437,E2 25724.437} C_VEL
LIN {X 0,Y 557.324,Z 781.393,A -85,B 0,C 180,E1 25723.103,E2 25723.103} C_VEL
LIN {X 0,Y 558.345,Z 764.302,A -85,B 0,C 180,E1 25721.898,E2 25721.898} C_VEL
LIN {X 0,Y 559.387,Z 746.229,A -85,B 0,C 180,E1 25720.852,E2 25720.852} C_VEL
LIN {X 0,Y 560.404,Z 727.196,A -85,B 0,C 180,E1 25719.966,E2 25719.966} C_VEL
LIN {X 0,Y 561.312,Z 707.248,A -85,B 0,C 180,E1 25719.244,E2 25719.244} C_VEL
LIN {X 0,Y 562.113,Z 686.328,A -85,B 0,C 180,E1 25718.692,E2 25718.692} C_VEL
LIN {X 0,Y 562.84,Z 658.287,A -85,B 0,C 180,E1 25718.211,E2 25718.211} C_VEL
LIN {X 0,Y 567.175,Z 492.226,A -85,B 0,C 180,E1 25715.577,E2 25715.577} C_VEL
LIN {X 0,Y 562.977,Z 452.936,A -85,B 0,C 180,E1 25714.657,E2 25714.657} C_VEL
LIN {X 0,Y 566.015,Z 399.396,A -85,B 0,C 180,E1 25711.109,E2 25711.109} C_VEL
LIN {X 0,Y 569.239,Z 347.997,A -85,B 0,C 180,E1 25707.661,E2 25707.661} C_VEL
LIN {X 0,Y 572.877,Z 295.512,A -85,B 0,C 180,E1 25704.094,E2 25704.094} C_VEL
LIN {X 0,Y 574.654,Z 270.17,A -85,B 0,C 180,E1 25702.344,E2 25702.344} C_VEL
LIN {X 0,Y 566.144,Z 247.725,A -85,B 0,C 180,E1 25700.041,E2 25700.041} C_VEL
LIN {X 0,Y 557.334,Z 226.081,A -85,B 0,C 180,E1 25697.659,E2 25697.659} C_VEL
LIN {X 0,Y 553.502,Z 216.282,A -85,B 0,C 180,E1 25696.538,E2 25696.538} C_VEL
LIN {X 0,Y 553.485,Z 216.285,A -85,B 0,C 180,E1 25695.578,E2 25695.578} C_VEL
LIN {X 0,Y 554.05,Z 216.863,A -85,B 0,C 180,E1 25695.27,E2 25695.27} C_VEL
LIN {X 0,Y 555.877,Z 219.571,A -85,B 0,C 180,E1 25694.837,E2 25694.837} C_VEL
LIN {X 0,Y 557.069,Z 224.539,A -85,B 0,C 180,E1 25694.397,E2 25694.397} C_VEL
LIN {X 0,Y 557.226,Z 232.762,A -85,B 0,C 180,E1 25693.87,E2 25693.87} C_VEL
LIN {X 0,Y 557.162,Z 239.787,A -85,B 0,C 180,E1 25693.369,E2 25693.369} C_VEL
LIN {X 0,Y 557.809,Z 242.388,A -85,B 0,C 180,E1 25693.118,E2 25693.118} C_VEL
LIN {X 0,Y 565.222,Z 259.709,A -85,B 0,C 180,E1 25691.153,E2 25691.153} C_VEL
LIN {X 0,Y 573.102,Z 280.2,A -85,B 0,C 180,E1 25688.909,E2 25688.909} C_VEL
LIN {X 0,Y 574.177,Z 283.466,A -85,B 0,C 180,E1 25688.564,E2 25688.564} C_VEL
LIN {X 0,Y 573.407,Z 324.892,A -85,B 0,C 180,E1 25685.649,E2 25685.649} C_VEL
LIN {X 0,Y 573.395,Z 344.327,A -85,B 0,C 180,E1 25684.402,E2 25684.402} C_VEL
LIN {X 0,Y 571.91,Z 351.804,A -85,B 0,C 180,E1 25684.127,E2 25684.127} C_VEL
LIN {X 0,Y 569.501,Z 444.205,A -85,B 0,C 180,E1 25682.82,E2 25682.82} C_VEL
LIN {X 0,Y 566.346,Z 528.179,A -85,B 0,C 180,E1 25681.447,E2 25681.447} C_VEL
LIN {X 0,Y 562.151,Z 625.543,A -85,B 0,C 180,E1 25679.643,E2 25679.643} C_VEL
LIN {X 0,Y 561.324,Z 647.713,A -85,B 0,C 180,E1 25679.098,E2 25679.098} C_VEL
LIN {X 0,Y 560.201,Z 668.926,A -85,B 0,C 180,E1 25678.397,E2 25678.397} C_VEL
LIN {X 0,Y 558.83,Z 690.378,A -85,B 0,C 180,E1 25677.492,E2 25677.492} C_VEL
LIN {X 0,Y 557.263,Z 710.898,A -85,B 0,C 180,E1 25676.422,E2 25676.422} C_VEL
LIN {X 0,Y 555.654,Z 729.737,A -85,B 0,C 180,E1 25675.244,E2 25675.244} C_VEL
LIN {X 0,Y 553.907,Z 748.467,A -85,B 0,C 180,E1 25673.851,E2 25673.851} C_VEL
LIN {X 0,Y 552.205,Z 765.569,A -85,B 0,C 180,E1 25672.349,E2 25672.349} C_VEL
LIN {X 0,Y 550.615,Z 781.323,A -85,B 0,C 180,E1 25670.736,E2 25670.736} C_VEL
LIN {X 0,Y 549.096,Z 796.575,A -85,B 0,C 180,E1 25668.913,E2 25668.913} C_VEL
LIN {X 0,Y 547.846,Z 809.646,A -85,B 0,C 180,E1 25667.088,E2 25667.088} C_VEL
LIN {X 0,Y 546.736,Z 821.984,A -85,B 0,C 180,E1 25665.052,E2 25665.052} C_VEL
LIN {X 0,Y 545.887,Z 832.446,A -85,B 0,C 180,E1 25662.977,E2 25662.977} C_VEL
LIN {X 0,Y 545.295,Z 841.157,A -85,B 0,C 180,E1 25660.887,E2 25660.887} C_VEL
LIN {X 0,Y 544.893,Z 848.325,A -85,B 0,C 180,E1 25658.761,E2 25658.761} C_VEL
LIN {X 0,Y 544.655,Z 854.059,A -85,B 0,C 180,E1 25656.536,E2 25656.536} C_VEL
LIN {X 0,Y 544.52,Z 858.022,A -85,B 0,C 180,E1 25654.318,E2 25654.318} C_VEL
LIN {X 0,Y 544.463,Z 860.459,A -85,B 0,C 180,E1 25652,E2 25652} C_VEL
LIN {X 0,Y 544.452,Z 861.183,A -85,B 0,C 180,E1 25649.79,E2 25649.79} C_VEL
LIN {X 0,Y 544.46,Z 860.248,A -85,B 0,C 180,E1 25647.579,E2 25647.579} C_VEL
LIN {X 0,Y 544.532,Z 857.68,A -85,B 0,C 180,E1 25645.366,E2 25645.366} C_VEL
LIN {X 0,Y 544.661,Z 853.521,A -85,B 0,C 180,E1 25643.147,E2 25643.147} C_VEL
LIN {X 0,Y 544.921,Z 847.677,A -85,B 0,C 180,E1 25640.921,E2 25640.921} C_VEL
LIN {X 0,Y 545.39,Z 839.904,A -85,B 0,C 180,E1 25638.687,E2 25638.687} C_VEL
LIN {X 0,Y 545.984,Z 831.159,A -85,B 0,C 180,E1 25636.659,E2 25636.659} C_VEL
LIN {X 0,Y 546.898,Z 820.032,A -85,B 0,C 180,E1 25634.518,E2 25634.518} C_VEL
LIN {X 0,Y 547.993,Z 808.097,A -85,B 0,C 180,E1 25632.588,E2 25632.588} C_VEL
LIN {X 0,Y 549.373,Z 793.988,A -85,B 0,C 180,E1 25630.655,E2 25630.655} C_VEL
LIN {X 0,Y 550.946,Z 778.217,A -85,B 0,C 180,E1 25628.829,E2 25628.829} C_VEL
LIN {X 0,Y 552.578,Z 761.895,A -85,B 0,C 180,E1 25627.218,E2 25627.218} C_VEL
LIN {X 0,Y 554.315,Z 744.086,A -85,B 0,C 180,E1 25625.715,E2 25625.715} C_VEL
LIN {X 0,Y 556.041,Z 725.374,A -85,B 0,C 180,E1 25624.375,E2 25624.375} C_VEL
LIN {X 0,Y 557.617,Z 706.84,A -85,B 0,C 180,E1 25623.251,E2 25623.251} C_VEL
LIN {X 0,Y 559.211,Z 685.417,A -85,B 0,C 180,E1 25622.181,E2 25622.181} C_VEL
LIN {X 0,Y 560.53,Z 663.88,A -85,B 0,C 180,E1 25621.324,E2 25621.324} C_VEL
LIN {X 0,Y 561.551,Z 642.269,A -85,B 0,C 180,E1 25620.66,E2 25620.66} C_VEL
LIN {X 0,Y 562.531,Z 615.38,A -85,B 0,C 180,E1 25620.064,E2 25620.064} C_VEL
LIN {X 0,Y 566.732,Z 519.503,A -85,B 0,C 180,E1 25618.31,E2 25618.31} C_VEL
LIN {X 0,Y 569.737,Z 437.707,A -85,B 0,C 180,E1 25616.99,E2 25616.99} C_VEL
LIN {X 0,Y 572.056,Z 350.5,A -85,B 0,C 180,E1 25615.749,E2 25615.749} C_VEL
LIN {X 0,Y 573.59,Z 342.93,A -85,B 0,C 180,E1 25615.43,E2 25615.43} C_VEL
LIN {X 0,Y 573.621,Z 308.086,A -85,B 0,C 180,E1 25613.1,E2 25613.1} C_VEL
LIN {X 0,Y 574.174,Z 282.895,A -85,B 0,C 180,E1 25611.276,E2 25611.276} C_VEL
LIN {X 0,Y 565.522,Z 260.216,A -85,B 0,C 180,E1 25608.792,E2 25608.792} C_VEL
LIN {X 0,Y 557.598,Z 241.874,A -85,B 0,C 180,E1 25606.723,E2 25606.723} C_VEL
LIN {X 0,Y 549.846,Z 226.072,A -85,B 0,C 180,E1 25604.876,E2 25604.876} C_VEL
LIN {X 0,Y 547.147,Z 221.142,A -85,B 0,C 180,E1 25604.274,E2 25604.274} C_VEL
LIN {X 0,Y 545.636,Z 217.747,A -85,B 0,C 180,E1 25603.899,E2 25603.899} C_VEL
LIN {X 0,Y 545.561,Z 217.262,A -85,B 0,C 180,E1 25603.852,E2 25603.852} C_VEL
LIN {X 0,Y 545.556,Z 217.26,A -85,B 0,C 180,E1 25600.452,E2 25600.452} C_VEL
LIN {X 0,Y 545.548,Z 217.257,A -85,B 0,C 180,E1 25597.085,E2 25597.085} C_VEL
LIN {X 0,Y 545.557,Z 217.259,A -85,B 0,C 180,E1 25593.687,E2 25593.687} C_VEL
LIN {X 0,Y 545.571,Z 217.27,A -85,B 0,C 180,E1 25590.265,E2 25590.265} C_VEL
LIN {X 0,Y 545.55,Z 217.267,A -85,B 0,C 180,E1 25586.8,E2 25586.8} C_VEL
LIN {X 0,Y 545.557,Z 217.242,A -85,B 0,C 180,E1 25583.436,E2 25583.436} C_VEL
LIN {X 0,Y 545.555,Z 217.265,A -85,B 0,C 180,E1 25580.044,E2 25580.044} C_VEL
LIN {X 0,Y 545.552,Z 217.256,A -85,B 0,C 180,E1 25576.614,E2 25576.614} C_VEL
LIN {X 0,Y 545.558,Z 217.251,A -85,B 0,C 180,E1 25573.244,E2 25573.244} C_VEL
LIN {X 0,Y 545.548,Z 217.274,A -85,B 0,C 180,E1 25569.814,E2 25569.814} C_VEL
LIN {X 0,Y 545.557,Z 217.241,A -85,B 0,C 180,E1 25566.419,E2 25566.419} C_VEL
LIN {X 0,Y 545.559,Z 217.27,A -85,B 0,C 180,E1 25562.942,E2 25562.942} C_VEL
LIN {X 0,Y 545.535,Z 217.238,A -85,B 0,C 180,E1 25559.58,E2 25559.58} C_VEL
LIN {X 0,Y 545.559,Z 217.276,A -85,B 0,C 180,E1 25556.217,E2 25556.217} C_VEL
LIN {X 0,Y 545.568,Z 217.234,A -85,B 0,C 180,E1 25552.841,E2 25552.841} C_VEL
LIN {X 0,Y 545.535,Z 217.274,A -85,B 0,C 180,E1 25549.439,E2 25549.439} C_VEL
LIN {X 0,Y 545.554,Z 217.276,A -85,B 0,C 180,E1 25545.999,E2 25545.999} C_VEL
LIN {X 0,Y 545.566,Z 217.273,A -85,B 0,C 180,E1 25542.618,E2 25542.618} C_VEL
LIN {X 0,Y 545.531,Z 217.273,A -85,B 0,C 180,E1 25539.283,E2 25539.283} C_VEL
LIN {X 0,Y 545.544,Z 217.269,A -85,B 0,C 180,E1 25535.875,E2 25535.875} C_VEL
LIN {X 0,Y 545.569,Z 217.267,A -85,B 0,C 180,E1 25532.493,E2 25532.493} C_VEL
LIN {X 0,Y 545.524,Z 217.277,A -85,B 0,C 180,E1 25529.244,E2 25529.244} C_VEL
LIN {X 0,Y 545.543,Z 217.269,A -85,B 0,C 180,E1 25525.885,E2 25525.885} C_VEL
LIN {X 0,Y 545.572,Z 217.42,A -85,B 0,C 180,E1 25523.998,E2 25523.998} C_VEL
LIN {X 0,Y 546.946,Z 220.925,A -85,B 0,C 180,E1 25523.548,E2 25523.548} C_VEL
LIN {X 0,Y 548.095,Z 223.012,A -85,B 0,C 180,E1 25523.246,E2 25523.246} C_VEL
LIN {X 0,Y 552.553,Z 231.732,A -85,B 0,C 180,E1 25522.029,E2 25522.029} C_VEL
LIN {X 0,Y 562.666,Z 251.502,A -85,B 0,C 180,E1 25519.428,E2 25519.428} C_VEL
LIN {X 0,Y 575.207,Z 277.134,A -85,B 0,C 180,E1 25516.361,E2 25516.361} C_VEL
LIN {X 0,Y 581.285,Z 289.975,A -85,B 0,C 180,E1 25514.94,E2 25514.94} C_VEL
LIN {X 0,Y 579.224,Z 311.616,A -85,B 0,C 180,E1 25513.699,E2 25513.699} C_VEL
LIN {X 0,Y 582.067,Z 336.568,A -85,B 0,C 180,E1 25513.055,E2 25513.055} C_VEL
LIN {X 0,Y 575.098,Z 576.403,A -85,B 0,C 180,E1 25509.55,E2 25509.55} C_VEL
LIN {X 0,Y 572.164,Z 692.789,A -85,B 0,C 180,E1 25507.889,E2 25507.889} C_VEL
LIN {X 0,Y 570.889,Z 717.376,A -85,B 0,C 180,E1 25507.368,E2 25507.368} C_VEL
LIN {X 0,Y 569.353,Z 740.821,A -85,B 0,C 180,E1 25506.71,E2 25506.71} C_VEL
LIN {X 0,Y 567.45,Z 764.117,A -85,B 0,C 180,E1 25505.866,E2 25505.866} C_VEL
LIN {X 0,Y 565.393,Z 786.321,A -85,B 0,C 180,E1 25504.897,E2 25504.897} C_VEL
LIN {X 0,Y 563.033,Z 808.895,A -85,B 0,C 180,E1 25503.699,E2 25503.699} C_VEL
LIN {X 0,Y 560.642,Z 830.726,A -85,B 0,C 180,E1 25502.347,E2 25502.347} C_VEL
LIN {X 0,Y 558.234,Z 850.811,A -85,B 0,C 180,E1 25500.881,E2 25500.881} C_VEL
LIN {X 0,Y 555.877,Z 870.326,A -85,B 0,C 180,E1 25499.261,E2 25499.261} C_VEL
LIN {X 0,Y 553.596,Z 888.677,A -85,B 0,C 180,E1 25497.483,E2 25497.483} C_VEL
LIN {X 0,Y 551.489,Z 906.198,A -85,B 0,C 180,E1 25495.563,E2 25495.563} C_VEL
LIN {X 0,Y 549.661,Z 921.747,A -85,B 0,C 180,E1 25493.591,E2 25493.591} C_VEL
LIN {X 0,Y 548.068,Z 936.356,A -85,B 0,C 180,E1 25491.496,E2 25491.496} C_VEL
LIN {X 0,Y 546.725,Z 949.932,A -85,B 0,C 180,E1 25489.22,E2 25489.22} C_VEL
LIN {X 0,Y 545.711,Z 961.807,A -85,B 0,C 180,E1 25486.938,E2 25486.938} C_VEL
LIN {X 0,Y 544.968,Z 972.165,A -85,B 0,C 180,E1 25484.558,E2 25484.558} C_VEL
LIN {X 0,Y 544.478,Z 980.864,A -85,B 0,C 180,E1 25482.192,E2 25482.192} C_VEL
LIN {X 0,Y 544.195,Z 988.079,A -85,B 0,C 180,E1 25479.732,E2 25479.732} C_VEL
LIN {X 0,Y 544.033,Z 992.996,A -85,B 0,C 180,E1 25477.604,E2 25477.604} C_VEL
LIN {X 0,Y 543.977,Z 997.187,A -85,B 0,C 180,E1 25475.167,E2 25475.167} C_VEL
LIN {X 0,Y 543.972,Z 999.563,A -85,B 0,C 180,E1 25472.845,E2 25472.845} C_VEL
LIN {X 0,Y 543.978,Z 1000.543,A -85,B 0,C 180,E1 25470.737,E2 25470.737} C_VEL
LIN {X 0,Y 543.995,Z 1000.31,A -85,B 0,C 180,E1 25468.42,E2 25468.42} C_VEL
LIN {X 0,Y 544.008,Z 998.31,A -85,B 0,C 180,E1 25465.889,E2 25465.889} C_VEL
LIN {X 0,Y 544.031,Z 995.184,A -85,B 0,C 180,E1 25463.669,E2 25463.669} C_VEL
LIN {X 0,Y 544.125,Z 989.937,A -85,B 0,C 180,E1 25461.12,E2 25461.12} C_VEL
LIN {X 0,Y 544.338,Z 983.75,A -85,B 0,C 180,E1 25458.879,E2 25458.879} C_VEL
LIN {X 0,Y 544.735,Z 975.699,A -85,B 0,C 180,E1 25456.519,E2 25456.519} C_VEL
LIN {X 0,Y 545.341,Z 965.751,A -85,B 0,C 180,E1 25454.146,E2 25454.146} C_VEL
LIN {X 0,Y 546.105,Z 955.604,A -85,B 0,C 180,E1 25452.085,E2 25452.085} C_VEL
LIN {X 0,Y 547.279,Z 941.8,A -85,B 0,C 180,E1 25449.688,E2 25449.688} C_VEL
LIN {X 0,Y 548.498,Z 928.642,A -85,B 0,C 180,E1 25447.717,E2 25447.717} C_VEL
LIN {X 0,Y 550.212,Z 911.802,A -85,B 0,C 180,E1 25445.522,E2 25445.522} C_VEL
LIN {X 0,Y 551.836,Z 896.243,A -85,B 0,C 180,E1 25443.755,E2 25443.755} C_VEL
LIN {X 0,Y 553.947,Z 876.817,A -85,B 0,C 180,E1 25441.823,E2 25441.823} C_VEL
LIN {X 0,Y 555.851,Z 859.161,A -85,B 0,C 180,E1 25440.292,E2 25440.292} C_VEL
LIN {X 0,Y 558.218,Z 836.465,A -85,B 0,C 180,E1 25438.584,E2 25438.584} C_VEL
LIN {X 0,Y 560.236,Z 816.516,A -85,B 0,C 180,E1 25437.293,E2 25437.293} C_VEL
LIN {X 0,Y 562.292,Z 794.189,A -85,B 0,C 180,E1 25436.057,E2 25436.057} C_VEL
LIN {X 0,Y 564.081,Z 773.206,A -85,B 0,C 180,E1 25435.072,E2 25435.072} C_VEL
LIN {X 0,Y 565.884,Z 749.209,A -85,B 0,C 180,E1 25434.144,E2 25434.144} C_VEL
LIN {X 0,Y 567.361,Z 726.472,A -85,B 0,C 180,E1 25433.439,E2 25433.439} C_VEL
LIN {X 0,Y 568.594,Z 702.091,A -85,B 0,C 180,E1 25432.871,E2 25432.871} C_VEL
LIN {X 0,Y 569.338,Z 679.341,A -85,B 0,C 180,E1 25432.488,E2 25432.488} C_VEL
LIN {X 0,Y 571.757,Z 561.36,A -85,B 0,C 180,E1 25430.854,E2 25430.854} C_VEL
LIN {X 0,Y 574.925,Z 458.823,A -85,B 0,C 180,E1 25429.273,E2 25429.273} C_VEL
LIN {X 0,Y 579.149,Z 367.753,A -85,B 0,C 180,E1 25427.734,E2 25427.734} C_VEL
LIN {X 0,Y 581.054,Z 335.093,A -85,B 0,C 180,E1 25427.145,E2 25427.145} C_VEL
LIN {X 0,Y 587.23,Z 314.419,A -85,B 0,C 180,E1 25425.516,E2 25425.516} C_VEL
LIN {X 0,Y 592.696,Z 300.447,A -85,B 0,C 180,E1 25424.301,E2 25424.301} C_VEL
LIN {X 0,Y 592.266,Z 297.133,A -85,B 0,C 180,E1 25423.137,E2 25423.137} C_VEL
LIN {X 0,Y 592.264,Z 295.324,A -85,B 0,C 180,E1 25421.825,E2 25421.825} C_VEL
LIN {X 0,Y 591.776,Z 297.266,A -85,B 0,C 180,E1 25420.326,E2 25420.326} C_VEL
LIN {X 0,Y 591.615,Z 299.404,A -85,B 0,C 180,E1 25419.581,E2 25419.581} C_VEL
LIN {X 0,Y 584.152,Z 317.161,A -85,B 0,C 180,E1 25417.792,E2 25417.792} C_VEL
LIN {X 0,Y 576.831,Z 341.117,A -85,B 0,C 180,E1 25415.561,E2 25415.561} C_VEL
LIN {X 0,Y 570.306,Z 371.749,A -85,B 0,C 180,E1 25412.923,E2 25412.923} C_VEL
LIN {X 0,Y 564.785,Z 407.956,A -85,B 0,C 180,E1 25410.026,E2 25410.026} C_VEL
LIN {X 0,Y 567.185,Z 438.405,A -85,B 0,C 180,E1 25408.603,E2 25408.603} C_VEL
LIN {X 0,Y 569.308,Z 473.337,A -85,B 0,C 180,E1 25407.217,E2 25407.217} C_VEL
LIN {X 0,Y 570.357,Z 498.769,A -85,B 0,C 180,E1 25406.343,E2 25406.343} C_VEL
LIN {X 0,Y 562.703,Z 603.388,A -85,B 0,C 180,E1 25404.074,E2 25404.074} C_VEL
LIN {X 0,Y 557.941,Z 688.582,A -85,B 0,C 180,E1 25402.263,E2 25402.263} C_VEL
LIN {X 0,Y 556.623,Z 711.497,A -85,B 0,C 180,E1 25401.583,E2 25401.583} C_VEL
LIN {X 0,Y 555.349,Z 732.232,A -85,B 0,C 180,E1 25400.775,E2 25400.775} C_VEL
LIN {X 0,Y 554.022,Z 752.678,A -85,B 0,C 180,E1 25399.779,E2 25399.779} C_VEL
LIN {X 0,Y 552.772,Z 771.115,A -85,B 0,C 180,E1 25398.673,E2 25398.673} C_VEL
LIN {X 0,Y 551.484,Z 789.197,A -85,B 0,C 180,E1 25397.353,E2 25397.353} C_VEL
LIN {X 0,Y 550.312,Z 804.791,A -85,B 0,C 180,E1 25395.978,E2 25395.978} C_VEL
LIN {X 0,Y 549.264,Z 818.297,A -85,B 0,C 180,E1 25394.55,E2 25394.55} C_VEL
LIN {X 0,Y 548.289,Z 830.809,A -85,B 0,C 180,E1 25392.962,E2 25392.962} C_VEL
LIN {X 0,Y 547.421,Z 841.703,A -85,B 0,C 180,E1 25391.271,E2 25391.271} C_VEL
LIN {X 0,Y 546.686,Z 850.984,A -85,B 0,C 180,E1 25389.475,E2 25389.475} C_VEL
LIN {X 0,Y 546.133,Z 858.24,A -85,B 0,C 180,E1 25387.681,E2 25387.681} C_VEL
LIN {X 0,Y 545.712,Z 863.903,A -85,B 0,C 180,E1 25385.784,E2 25385.784} C_VEL
LIN {X 0,Y 545.397,Z 867.699,A -85,B 0,C 180,E1 25383.89,E2 25383.89} C_VEL
LIN {X 0,Y 545.189,Z 869.735,A -85,B 0,C 180,E1 25381.997,E2 25381.997} C_VEL
LIN {X 0,Y 545.062,Z 870.008,A -85,B 0,C 180,E1 25380,E2 25380} C_VEL
LIN {X 0,Y 544.997,Z 868.394,A -85,B 0,C 180,E1 25378.002,E2 25378.002} C_VEL
LIN {X 0,Y 545.022,Z 865.153,A -85,B 0,C 180,E1 25376.108,E2 25376.108} C_VEL
LIN {X 0,Y 545.145,Z 860.169,A -85,B 0,C 180,E1 25374.21,E2 25374.21} C_VEL
LIN {X 0,Y 545.37,Z 853.329,A -85,B 0,C 180,E1 25372.308,E2 25372.308} C_VEL
LIN {X 0,Y 545.733,Z 845.011,A -85,B 0,C 180,E1 25370.509,E2 25370.509} C_VEL
LIN {X 0,Y 546.275,Z 834.634,A -85,B 0,C 180,E1 25368.706,E2 25368.706} C_VEL
LIN {X 0,Y 546.971,Z 822.697,A -85,B 0,C 180,E1 25367.006,E2 25367.006} C_VEL
LIN {X 0,Y 547.817,Z 809.197,A -85,B 0,C 180,E1 25365.411,E2 25365.411} C_VEL
LIN {X 0,Y 548.794,Z 794.082,A -85,B 0,C 180,E1 25363.922,E2 25363.922} C_VEL
LIN {X 0,Y 549.884,Z 777.199,A -85,B 0,C 180,E1 25362.54,E2 25362.54} C_VEL
LIN {X 0,Y 550.942,Z 759.953,A -85,B 0,C 180,E1 25361.372,E2 25361.372} C_VEL
LIN {X 0,Y 552.012,Z 741.997,A -85,B 0,C 180,E1 25360.374,E2 25360.374} C_VEL
LIN {X 0,Y 553.037,Z 722.914,A -85,B 0,C 180,E1 25359.522,E2 25359.522} C_VEL
LIN {X 0,Y 553.969,Z 702.7,A -85,B 0,C 180,E1 25358.825,E2 25358.825} C_VEL
LIN {X 0,Y 554.788,Z 681.509,A -85,B 0,C 180,E1 25358.303,E2 25358.303} C_VEL
LIN {X 0,Y 559.864,Z 492.751,A -85,B 0,C 180,E1 25355.237,E2 25355.237} C_VEL
LIN {X 0,Y 555.561,Z 452.559,A -85,B 0,C 180,E1 25354.294,E2 25354.294} C_VEL
LIN {X 0,Y 558.757,Z 398.884,A -85,B 0,C 180,E1 25350.697,E2 25350.697} C_VEL
LIN {X 0,Y 562.093,Z 348.261,A -85,B 0,C 180,E1 25347.263,E2 25347.263} C_VEL
LIN {X 0,Y 565.901,Z 296.072,A -85,B 0,C 180,E1 25343.679,E2 25343.679} C_VEL
LIN {X 0,Y 567.638,Z 273.459,A -85,B 0,C 180,E1 25342.106,E2 25342.106} C_VEL
LIN {X 0,Y 559.201,Z 250.997,A -85,B 0,C 180,E1 25339.774,E2 25339.774} C_VEL
LIN {X 0,Y 549.663,Z 227.521,A -85,B 0,C 180,E1 25337.147,E2 25337.147} C_VEL
LIN {X 0,Y 545.622,Z 217.809,A -85,B 0,C 180,E1 25335.991,E2 25335.991} C_VEL
LIN {X 0,Y 546.762,Z 220.631,A -85,B 0,C 180,E1 25335.686,E2 25335.686} C_VEL
LIN {X 0,Y 547.967,Z 222.455,A -85,B 0,C 180,E1 25335.444,E2 25335.444} C_VEL
LIN {X 0,Y 556.854,Z 240.409,A -85,B 0,C 180,E1 25333.346,E2 25333.346} C_VEL
LIN {X 0,Y 557.809,Z 242.388,A -85,B 0,C 180,E1 25333.118,E2 25333.118} C_VEL
LIN {X 0,Y 559.194,Z 248.018,A -85,B 0,C 180,E1 25332.587,E2 25332.587} C_VEL
LIN {X 0,Y 560.151,Z 264.918,A -85,B 0,C 180,E1 25331.269,E2 25331.269} C_VEL
LIN {X 0,Y 561.338,Z 269.652,A -85,B 0,C 180,E1 25330.803,E2 25330.803} C_VEL
LIN {X 0,Y 567.742,Z 287.266,A -85,B 0,C 180,E1 25328.882,E2 25328.882} C_VEL
LIN {X 0,Y 567.028,Z 328.039,A -85,B 0,C 180,E1 25326.022,E2 25326.022} C_VEL
LIN {X 0,Y 567.18,Z 345.277,A -85,B 0,C 180,E1 25324.901,E2 25324.901} C_VEL
LIN {X 0,Y 565.296,Z 354.489,A -85,B 0,C 180,E1 25324.555,E2 25324.555} C_VEL
LIN {X 0,Y 562.822,Z 445.712,A -85,B 0,C 180,E1 25323.252,E2 25323.252} C_VEL
LIN {X 0,Y 559.596,Z 528.217,A -85,B 0,C 180,E1 25321.886,E2 25321.886} C_VEL
LIN {X 0,Y 555.257,Z 623.232,A -85,B 0,C 180,E1 25320.097,E2 25320.097} C_VEL
LIN {X 0,Y 554.368,Z 646.878,A -85,B 0,C 180,E1 25319.528,E2 25319.528} C_VEL
LIN {X 0,Y 553.181,Z 669.205,A -85,B 0,C 180,E1 25318.797,E2 25318.797} C_VEL
LIN {X 0,Y 551.745,Z 690.945,A -85,B 0,C 180,E1 25317.876,E2 25317.876} C_VEL
LIN {X 0,Y 550.167,Z 710.976,A -85,B 0,C 180,E1 25316.828,E2 25316.828} C_VEL
LIN {X 0,Y 548.428,Z 730.474,A -85,B 0,C 180,E1 25315.601,E2 25315.601} C_VEL
LIN {X 0,Y 546.525,Z 749.886,A -85,B 0,C 180,E1 25314.136,E2 25314.136} C_VEL
LIN {X 0,Y 544.687,Z 767.505,A -85,B 0,C 180,E1 25312.561,E2 25312.561} C_VEL
LIN {X 0,Y 542.971,Z 783.58,A -85,B 0,C 180,E1 25310.875,E2 25310.875} C_VEL
LIN {X 0,Y 541.341,Z 799.064,A -85,B 0,C 180,E1 25308.971,E2 25308.971} C_VEL
LIN {X 0,Y 539.973,Z 812.571,A -85,B 0,C 180,E1 25307.012,E2 25307.012} C_VEL
LIN {X 0,Y 538.893,Z 824.057,A -85,B 0,C 180,E1 25305.056,E2 25305.056} C_VEL
LIN {X 0,Y 537.996,Z 834.666,A -85,B 0,C 180,E1 25302.887,E2 25302.887} C_VEL
LIN {X 0,Y 537.366,Z 843.29,A -85,B 0,C 180,E1 25300.724,E2 25300.724} C_VEL
LIN {X 0,Y 536.938,Z 850.477,A -85,B 0,C 180,E1 25298.46,E2 25298.46} C_VEL
LIN {X 0,Y 536.699,Z 855.899,A -85,B 0,C 180,E1 25296.203,E2 25296.203} C_VEL
LIN {X 0,Y 536.578,Z 859.644,A -85,B 0,C 180,E1 25293.954,E2 25293.954} C_VEL
LIN {X 0,Y 536.52,Z 861.661,A -85,B 0,C 180,E1 25291.709,E2 25291.709} C_VEL
LIN {X 0,Y 536.5,Z 862.115,A -85,B 0,C 180,E1 25289.466,E2 25289.466} C_VEL
LIN {X 0,Y 536.535,Z 861.09,A -85,B 0,C 180,E1 25287.311,E2 25287.311} C_VEL
LIN {X 0,Y 536.616,Z 858.351,A -85,B 0,C 180,E1 25285.083,E2 25285.083} C_VEL
LIN {X 0,Y 536.76,Z 853.991,A -85,B 0,C 180,E1 25282.83,E2 25282.83} C_VEL
LIN {X 0,Y 537.06,Z 848.228,A -85,B 0,C 180,E1 25280.663,E2 25280.663} C_VEL
LIN {X 0,Y 537.582,Z 840.447,A -85,B 0,C 180,E1 25278.412,E2 25278.412} C_VEL
LIN {X 0,Y 538.282,Z 831.066,A -85,B 0,C 180,E1 25276.245,E2 25276.245} C_VEL
LIN {X 0,Y 539.238,Z 820.299,A -85,B 0,C 180,E1 25274.182,E2 25274.182} C_VEL
LIN {X 0,Y 540.484,Z 807.46,A -85,B 0,C 180,E1 25272.116,E2 25272.116} C_VEL
LIN {X 0,Y 541.931,Z 793.541,A -85,B 0,C 180,E1 25270.217,E2 25270.217} C_VEL
LIN {X 0,Y 543.588,Z 778.05,A -85,B 0,C 180,E1 25268.415,E2 25268.415} C_VEL
LIN {X 0,Y 545.433,Z 760.64,A -85,B 0,C 180,E1 25266.699,E2 25266.699} C_VEL
LIN {X 0,Y 547.234,Z 742.771,A -85,B 0,C 180,E1 25265.207,E2 25265.207} C_VEL
LIN {X 0,Y 549.001,Z 724.32,A -85,B 0,C 180,E1 25263.9,E2 25263.9} C_VEL
LIN {X 0,Y 550.7,Z 704.388,A -85,B 0,C 180,E1 25262.712,E2 25262.712} C_VEL
LIN {X 0,Y 552.219,Z 684.621,A -85,B 0,C 180,E1 25261.739,E2 25261.739} C_VEL
LIN {X 0,Y 553.591,Z 663.149,A -85,B 0,C 180,E1 25260.886,E2 25260.886} C_VEL
LIN {X 0,Y 554.663,Z 640.615,A -85,B 0,C 180,E1 25260.203,E2 25260.203} C_VEL
LIN {X 0,Y 556.053,Z 605.062,A -85,B 0,C 180,E1 25259.449,E2 25259.449} C_VEL
LIN {X 0,Y 560.307,Z 512.148,A -85,B 0,C 180,E1 25257.741,E2 25257.741} C_VEL
LIN {X 0,Y 563.191,Z 435.44,A -85,B 0,C 180,E1 25256.499,E2 25256.499} C_VEL
LIN {X 0,Y 565.436,Z 353.224,A -85,B 0,C 180,E1 25255.322,E2 25255.322} C_VEL
LIN {X 0,Y 567.211,Z 344.978,A -85,B 0,C 180,E1 25254.985,E2 25254.985} C_VEL
LIN {X 0,Y 567.263,Z 309.602,A -85,B 0,C 180,E1 25252.617,E2 25252.617} C_VEL
LIN {X 0,Y 567.719,Z 286.667,A -85,B 0,C 180,E1 25250.96,E2 25250.96} C_VEL
LIN {X 0,Y 559.678,Z 265.46,A -85,B 0,C 180,E1 25248.621,E2 25248.621} C_VEL
LIN {X 0,Y 551.645,Z 246.659,A -85,B 0,C 180,E1 25246.467,E2 25246.467} C_VEL
LIN {X 0,Y 543.96,Z 231.051,A -85,B 0,C 180,E1 25244.603,E2 25244.603} C_VEL
LIN {X 0,Y 539.479,Z 222.458,A -85,B 0,C 180,E1 25243.557,E2 25243.557} C_VEL
LIN {X 0,Y 537.813,Z 219.316,A -85,B 0,C 180,E1 25243.171,E2 25243.171} C_VEL
LIN {X 0,Y 537.603,Z 218.255,A -85,B 0,C 180,E1 25243.046,E2 25243.046} C_VEL
LIN {X 0,Y 537.624,Z 218.253,A -85,B 0,C 180,E1 25239.649,E2 25239.649} C_VEL
LIN {X 0,Y 537.621,Z 218.247,A -85,B 0,C 180,E1 25236.179,E2 25236.179} C_VEL
LIN {X 0,Y 537.606,Z 218.241,A -85,B 0,C 180,E1 25232.768,E2 25232.768} C_VEL
LIN {X 0,Y 537.626,Z 218.247,A -85,B 0,C 180,E1 25229.406,E2 25229.406} C_VEL
LIN {X 0,Y 537.617,Z 218.262,A -85,B 0,C 180,E1 25225.917,E2 25225.917} C_VEL
LIN {X 0,Y 537.612,Z 218.238,A -85,B 0,C 180,E1 25222.528,E2 25222.528} C_VEL
LIN {X 0,Y 537.62,Z 218.24,A -85,B 0,C 180,E1 25219.107,E2 25219.107} C_VEL
LIN {X 0,Y 537.61,Z 218.26,A -85,B 0,C 180,E1 25215.645,E2 25215.645} C_VEL
LIN {X 0,Y 537.616,Z 218.228,A -85,B 0,C 180,E1 25212.241,E2 25212.241} C_VEL
LIN {X 0,Y 537.619,Z 218.261,A -85,B 0,C 180,E1 25208.772,E2 25208.772} C_VEL
LIN {X 0,Y 537.604,Z 218.231,A -85,B 0,C 180,E1 25205.443,E2 25205.443} C_VEL
LIN {X 0,Y 537.614,Z 218.259,A -85,B 0,C 180,E1 25202.025,E2 25202.025} C_VEL
LIN {X 0,Y 537.618,Z 218.229,A -85,B 0,C 180,E1 25198.615,E2 25198.615} C_VEL
LIN {X 0,Y 537.609,Z 218.258,A -85,B 0,C 180,E1 25195.199,E2 25195.199} C_VEL
LIN {X 0,Y 537.597,Z 218.237,A -85,B 0,C 180,E1 25191.766,E2 25191.766} C_VEL
LIN {X 0,Y 537.624,Z 218.262,A -85,B 0,C 180,E1 25188.413,E2 25188.413} C_VEL
LIN {X 0,Y 537.609,Z 218.258,A -85,B 0,C 180,E1 25185.017,E2 25185.017} C_VEL
LIN {X 0,Y 537.592,Z 218.257,A -85,B 0,C 180,E1 25181.567,E2 25181.567} C_VEL
LIN {X 0,Y 537.627,Z 218.256,A -85,B 0,C 180,E1 25178.133,E2 25178.133} C_VEL
LIN {X 0,Y 537.623,Z 218.261,A -85,B 0,C 180,E1 25174.673,E2 25174.673} C_VEL
LIN {X 0,Y 537.588,Z 218.263,A -85,B 0,C 180,E1 25171.323,E2 25171.323} C_VEL
LIN {X 0,Y 537.612,Z 218.258,A -85,B 0,C 180,E1 25167.99,E2 25167.99} C_VEL
LIN {X 0,Y 537.608,Z 218.319,A -85,B 0,C 180,E1 25164.856,E2 25164.856} C_VEL
LIN {X 0,Y 539.036,Z 221.888,A -85,B 0,C 180,E1 25164.376,E2 25164.376} C_VEL
LIN {X 0,Y 540.145,Z 223.959,A -85,B 0,C 180,E1 25164.068,E2 25164.068} C_VEL
LIN {X 0,Y 547.148,Z 237.722,A -85,B 0,C 180,E1 25162.135,E2 25162.135} C_VEL
LIN {X 0,Y 555.793,Z 254.685,A -85,B 0,C 180,E1 25159.87,E2 25159.87} C_VEL
LIN {X 0,Y 567.777,Z 279.06,A -85,B 0,C 180,E1 25156.898,E2 25156.898} C_VEL
LIN {X 0,Y 574.624,Z 293.591,A -85,B 0,C 180,E1 25155.266,E2 25155.266} C_VEL
LIN {X 0,Y 572.789,Z 312.388,A -85,B 0,C 180,E1 25154.181,E2 25154.181} C_VEL
LIN {X 0,Y 575.609,Z 337.913,A -85,B 0,C 180,E1 25153.511,E2 25153.511} C_VEL
LIN {X 0,Y 568.399,Z 574.17,A -85,B 0,C 180,E1 25150.013,E2 25150.013} C_VEL
LIN {X 0,Y 565.24,Z 692.907,A -85,B 0,C 180,E1 25148.293,E2 25148.293} C_VEL
LIN {X 0,Y 563.911,Z 717.312,A -85,B 0,C 180,E1 25147.769,E2 25147.769} C_VEL
LIN {X 0,Y 562.316,Z 740.745,A -85,B 0,C 180,E1 25147.102,E2 25147.102} C_VEL
LIN {X 0,Y 560.358,Z 763.761,A -85,B 0,C 180,E1 25146.259,E2 25146.259} C_VEL
LIN {X 0,Y 558.236,Z 785.814,A -85,B 0,C 180,E1 25145.285,E2 25145.285} C_VEL
LIN {X 0,Y 555.841,Z 808.023,A -85,B 0,C 180,E1 25144.101,E2 25144.101} C_VEL
LIN {X 0,Y 553.354,Z 829.831,A -85,B 0,C 180,E1 25142.744,E2 25142.744} C_VEL
LIN {X 0,Y 550.83,Z 850.208,A -85,B 0,C 180,E1 25141.242,E2 25141.242} C_VEL
LIN {X 0,Y 548.389,Z 869.628,A -85,B 0,C 180,E1 25139.612,E2 25139.612} C_VEL
LIN {X 0,Y 545.99,Z 888.123,A -85,B 0,C 180,E1 25137.805,E2 25137.805} C_VEL
LIN {X 0,Y 543.894,Z 904.929,A -85,B 0,C 180,E1 25135.947,E2 25135.947} C_VEL
LIN {X 0,Y 541.864,Z 921.378,A -85,B 0,C 180,E1 25133.836,E2 25133.836} C_VEL
LIN {X 0,Y 540.205,Z 936.094,A -85,B 0,C 180,E1 25131.693,E2 25131.693} C_VEL
LIN {X 0,Y 538.814,Z 949.512,A -85,B 0,C 180,E1 25129.401,E2 25129.401} C_VEL
LIN {X 0,Y 537.763,Z 961.35,A -85,B 0,C 180,E1 25127.084,E2 25127.084} C_VEL
LIN {X 0,Y 536.997,Z 971.653,A -85,B 0,C 180,E1 25124.669,E2 25124.669} C_VEL
LIN {X 0,Y 536.496,Z 980.32,A -85,B 0,C 180,E1 25122.267,E2 25122.267} C_VEL
LIN {X 0,Y 536.213,Z 987.47,A -85,B 0,C 180,E1 25119.77,E2 25119.77} C_VEL
LIN {X 0,Y 536.056,Z 992.559,A -85,B 0,C 180,E1 25117.502,E2 25117.502} C_VEL
LIN {X 0,Y 536.021,Z 996.702,A -85,B 0,C 180,E1 25114.922,E2 25114.922} C_VEL
LIN {X 0,Y 536.018,Z 998.855,A -85,B 0,C 180,E1 25112.673,E2 25112.673} C_VEL
LIN {X 0,Y 536.024,Z 999.722,A -85,B 0,C 180,E1 25110.534,E2 25110.534} C_VEL
LIN {X 0,Y 536.049,Z 999.206,A -85,B 0,C 180,E1 25107.969,E2 25107.969} C_VEL
LIN {X 0,Y 536.052,Z 997.162,A -85,B 0,C 180,E1 25105.614,E2 25105.614} C_VEL
LIN {X 0,Y 536.086,Z 993.523,A -85,B 0,C 180,E1 25103.144,E2 25103.144} C_VEL
LIN {X 0,Y 536.215,Z 987.846,A -85,B 0,C 180,E1 25100.554,E2 25100.554} C_VEL
LIN {X 0,Y 536.436,Z 981.355,A -85,B 0,C 180,E1 25098.277,E2 25098.277} C_VEL
LIN {X 0,Y 536.902,Z 972.446,A -85,B 0,C 180,E1 25095.769,E2 25095.769} C_VEL
LIN {X 0,Y 537.486,Z 963.529,A -85,B 0,C 180,E1 25093.686,E2 25093.686} C_VEL
LIN {X 0,Y 538.381,Z 952.034,A -85,B 0,C 180,E1 25091.371,E2 25091.371} C_VEL
LIN {X 0,Y 539.558,Z 938.995,A -85,B 0,C 180,E1 25089.157,E2 25089.157} C_VEL
LIN {X 0,Y 541.046,Z 924.362,A -85,B 0,C 180,E1 25086.976,E2 25086.976} C_VEL
LIN {X 0,Y 542.72,Z 908.339,A -85,B 0,C 180,E1 25084.929,E2 25084.929} C_VEL
LIN {X 0,Y 544.653,Z 891.221,A -85,B 0,C 180,E1 25082.997,E2 25082.997} C_VEL
LIN {X 0,Y 546.634,Z 873.266,A -85,B 0,C 180,E1 25081.244,E2 25081.244} C_VEL
LIN {X 0,Y 548.843,Z 853.871,A -85,B 0,C 180,E1 25079.571,E2 25079.571} C_VEL
LIN {X 0,Y 551.07,Z 833.524,A -85,B 0,C 180,E1 25078.068,E2 25078.068} C_VEL
LIN {X 0,Y 553.329,Z 811.96,A -85,B 0,C 180,E1 25076.678,E2 25076.678} C_VEL
LIN {X 0,Y 555.351,Z 790.52,A -85,B 0,C 180,E1 25075.511,E2 25075.511} C_VEL
LIN {X 0,Y 557.466,Z 767.194,A -85,B 0,C 180,E1 25074.438,E2 25074.438} C_VEL
LIN {X 0,Y 559.208,Z 744.36,A -85,B 0,C 180,E1 25073.585,E2 25073.585} C_VEL
LIN {X 0,Y 560.836,Z 719.263,A -85,B 0,C 180,E1 25072.844,E2 25072.844} C_VEL
LIN {X 0,Y 561.925,Z 697.13,A -85,B 0,C 180,E1 25072.353,E2 25072.353} C_VEL
LIN {X 0,Y 562.89,Z 662.167,A -85,B 0,C 180,E1 25071.823,E2 25071.823} C_VEL
LIN {X 0,Y 565.438,Z 555.973,A -85,B 0,C 180,E1 25070.298,E2 25070.298} C_VEL
LIN {X 0,Y 568.875,Z 459.993,A -85,B 0,C 180,E1 25068.758,E2 25068.758} C_VEL
LIN {X 0,Y 573.522,Z 371.719,A -85,B 0,C 180,E1 25067.213,E2 25067.213} C_VEL
LIN {X 0,Y 575.928,Z 337.583,A -85,B 0,C 180,E1 25066.567,E2 25066.567} C_VEL
LIN {X 0,Y 582.392,Z 318.422,A -85,B 0,C 180,E1 25065.02,E2 25065.02} C_VEL
LIN {X 0,Y 587.759,Z 305.833,A -85,B 0,C 180,E1 25063.908,E2 25063.908} C_VEL
LIN {X 0,Y 587.512,Z 303.318,A -85,B 0,C 180,E1 25062.904,E2 25062.904} C_VEL
LIN {X 0,Y 587.613,Z 301.92,A -85,B 0,C 180,E1 25061.814,E2 25061.814} C_VEL
LIN {X 0,Y 587.057,Z 303.686,A -85,B 0,C 180,E1 25060.417,E2 25060.417} C_VEL
LIN {X 0,Y 586.853,Z 304.967,A -85,B 0,C 180,E1 25059.967,E2 25059.967} C_VEL
LIN {X 0,Y 578.996,Z 322.192,A -85,B 0,C 180,E1 25058.188,E2 25058.188} C_VEL
LIN {X 0,Y 571.699,Z 343.811,A -85,B 0,C 180,E1 25056.115,E2 25056.115} C_VEL
LIN {X 0,Y 564.744,Z 372.896,A -85,B 0,C 180,E1 25053.532,E2 25053.532} C_VEL
LIN {X 0,Y 559.333,Z 404.006,A -85,B 0,C 180,E1 25050.965,E2 25050.965} C_VEL
LIN {X 0,Y 561.123,Z 431.011,A -85,B 0,C 180,E1 25049.604,E2 25049.604} C_VEL
LIN {X 0,Y 562.74,Z 458.292,A -85,B 0,C 180,E1 25048.414,E2 25048.414} C_VEL
LIN {X 0,Y 564.237,Z 492.411,A -85,B 0,C 180,E1 25047.115,E2 25047.115} C_VEL
LIN {X 0,Y 564.296,Z 500.86,A -85,B 0,C 180,E1 25046.848,E2 25046.848} C_VEL
LIN {X 0,Y 555.896,Z 607.992,A -85,B 0,C 180,E1 25044.455,E2 25044.455} C_VEL
LIN {X 0,Y 550.995,Z 689.896,A -85,B 0,C 180,E1 25042.658,E2 25042.658} C_VEL
LIN {X 0,Y 549.559,Z 712.618,A -85,B 0,C 180,E1 25041.956,E2 25041.956} C_VEL
LIN {X 0,Y 548.102,Z 734.86,A -85,B 0,C 180,E1 25041.062,E2 25041.062} C_VEL
LIN {X 0,Y 546.7,Z 754.813,A -85,B 0,C 180,E1 25040.056,E2 25040.056} C_VEL
LIN {X 0,Y 545.257,Z 774.457,A -85,B 0,C 180,E1 25038.829,E2 25038.829} C_VEL
LIN {X 0,Y 544.007,Z 790.835,A -85,B 0,C 180,E1 25037.598,E2 25037.598} C_VEL
LIN {X 0,Y 542.76,Z 806.281,A -85,B 0,C 180,E1 25036.206,E2 25036.206} C_VEL
LIN {X 0,Y 541.656,Z 819.766,A -85,B 0,C 180,E1 25034.759,E2 25034.759} C_VEL
LIN {X 0,Y 540.606,Z 832.173,A -85,B 0,C 180,E1 25033.15,E2 25033.15} C_VEL
LIN {X 0,Y 539.697,Z 842.932,A -85,B 0,C 180,E1 25031.457,E2 25031.457} C_VEL
LIN {X 0,Y 538.942,Z 851.839,A -85,B 0,C 180,E1 25029.72,E2 25029.72} C_VEL
LIN {X 0,Y 538.33,Z 859.145,A -85,B 0,C 180,E1 25027.9,E2 25027.9} C_VEL
LIN {X 0,Y 537.866,Z 864.892,A -85,B 0,C 180,E1 25025.976,E2 25025.976} C_VEL
LIN {X 0,Y 537.517,Z 868.74,A -85,B 0,C 180,E1 25024.053,E2 25024.053} C_VEL
LIN {X 0,Y 537.273,Z 870.862,A -85,B 0,C 180,E1 25022.026,E2 25022.026} C_VEL
LIN {X 0,Y 537.137,Z 871.108,A -85,B 0,C 180,E1 25020.107,E2 25020.107} C_VEL
LIN {X 0,Y 537.062,Z 869.527,A -85,B 0,C 180,E1 25018.08,E2 25018.08} C_VEL
LIN {X 0,Y 537.085,Z 866.053,A -85,B 0,C 180,E1 25016.05,E2 25016.05} C_VEL
LIN {X 0,Y 537.214,Z 860.974,A -85,B 0,C 180,E1 25014.124,E2 25014.124} C_VEL
LIN {X 0,Y 537.453,Z 854.029,A -85,B 0,C 180,E1 25012.194,E2 25012.194} C_VEL
LIN {X 0,Y 537.835,Z 845.598,A -85,B 0,C 180,E1 25010.368,E2 25010.368} C_VEL
LIN {X 0,Y 538.407,Z 835.101,A -85,B 0,C 180,E1 25008.538,E2 25008.538} C_VEL
LIN {X 0,Y 539.138,Z 823.039,A -85,B 0,C 180,E1 25006.814,E2 25006.814} C_VEL
LIN {X 0,Y 540.025,Z 809.408,A -85,B 0,C 180,E1 25005.196,E2 25005.196} C_VEL
LIN {X 0,Y 541.048,Z 794.154,A -85,B 0,C 180,E1 25003.686,E2 25003.686} C_VEL
LIN {X 0,Y 542.144,Z 777.833,A -85,B 0,C 180,E1 25002.338,E2 25002.338} C_VEL
LIN {X 0,Y 543.242,Z 760.571,A -85,B 0,C 180,E1 25001.154,E2 25001.154} C_VEL
LIN {X 0,Y 544.376,Z 742.252,A -85,B 0,C 180,E1 25000.123,E2 25000.123} C_VEL
LIN {X 0,Y 545.486,Z 722.321,A -85,B 0,C 180,E1 24999.225,E2 24999.225} C_VEL
LIN {X 0,Y 546.474,Z 701.565,A -85,B 0,C 180,E1 24998.51,E2 24998.51} C_VEL
LIN {X 0,Y 547.309,Z 680.19,A -85,B 0,C 180,E1 24997.991,E2 24997.991} C_VEL
LIN {X 0,Y 552.595,Z 493.47,A -85,B 0,C 180,E1 24994.893,E2 24994.893} C_VEL
LIN {X 0,Y 548.2,Z 451.265,A -85,B 0,C 180,E1 24993.865,E2 24993.865} C_VEL
LIN {X 0,Y 551.51,Z 398.377,A -85,B 0,C 180,E1 24990.277,E2 24990.277} C_VEL
LIN {X 0,Y 554.973,Z 348.44,A -85,B 0,C 180,E1 24986.851,E2 24986.851} C_VEL
LIN {X 0,Y 558.933,Z 296.84,A -85,B 0,C 180,E1 24983.268,E2 24983.268} C_VEL
LIN {X 0,Y 560.457,Z 276.111,A -85,B 0,C 180,E1 24981.802,E2 24981.802} C_VEL
LIN {X 0,Y 552.254,Z 254.309,A -85,B 0,C 180,E1 24979.503,E2 24979.503} C_VEL
LIN {X 0,Y 543.152,Z 231.849,A -85,B 0,C 180,E1 24976.957,E2 24976.957} C_VEL
LIN {X 0,Y 540.134,Z 224.771,A -85,B 0,C 180,E1 24976.11,E2 24976.11} C_VEL
LIN {X 0,Y 542.145,Z 227.323,A -85,B 0,C 180,E1 24975.727,E2 24975.727} C_VEL
LIN {X 0,Y 551.923,Z 247.289,A -85,B 0,C 180,E1 24973.356,E2 24973.356} C_VEL
LIN {X 0,Y 560.18,Z 266.792,A -85,B 0,C 180,E1 24971.127,E2 24971.127} C_VEL
LIN {X 0,Y 561.338,Z 269.652,A -85,B 0,C 180,E1 24970.803,E2 24970.803} C_VEL
LIN {X 0,Y 562.612,Z 275.26,A -85,B 0,C 180,E1 24970.269,E2 24970.269} C_VEL
LIN {X 0,Y 562.528,Z 283.43,A -85,B 0,C 180,E1 24969.667,E2 24969.667} C_VEL
LIN {X 0,Y 561.17,Z 298.745,A -85,B 0,C 180,E1 24968.658,E2 24968.658} C_VEL
LIN {X 0,Y 560.711,Z 337.616,A -85,B 0,C 180,E1 24965.979,E2 24965.979} C_VEL
LIN {X 0,Y 560.705,Z 347.467,A -85,B 0,C 180,E1 24965.357,E2 24965.357} C_VEL
LIN {X 0,Y 558.715,Z 357.173,A -85,B 0,C 180,E1 24964.994,E2 24964.994} C_VEL
LIN {X 0,Y 556.167,Z 447.442,A -85,B 0,C 180,E1 24963.692,E2 24963.692} C_VEL
LIN {X 0,Y 552.932,Z 527.219,A -85,B 0,C 180,E1 24962.355,E2 24962.355} C_VEL
LIN {X 0,Y 548.547,Z 618.27,A -85,B 0,C 180,E1 24960.617,E2 24960.617} C_VEL
LIN {X 0,Y 547.462,Z 645.913,A -85,B 0,C 180,E1 24959.976,E2 24959.976} C_VEL
LIN {X 0,Y 546.334,Z 667.535,A -85,B 0,C 180,E1 24959.283,E2 24959.283} C_VEL
LIN {X 0,Y 544.964,Z 688.15,A -85,B 0,C 180,E1 24958.433,E2 24958.433} C_VEL
LIN {X 0,Y 543.313,Z 708.436,A -85,B 0,C 180,E1 24957.393,E2 24957.393} C_VEL
LIN {X 0,Y 541.53,Z 727.919,A -85,B 0,C 180,E1 24956.186,E2 24956.186} C_VEL
LIN {X 0,Y 539.576,Z 747.236,A -85,B 0,C 180,E1 24954.759,E2 24954.759} C_VEL
LIN {X 0,Y 537.609,Z 765.448,A -85,B 0,C 180,E1 24953.164,E2 24953.164} C_VEL
LIN {X 0,Y 535.836,Z 781.469,A -85,B 0,C 180,E1 24951.518,E2 24951.518} C_VEL
LIN {X 0,Y 534.13,Z 796.811,A -85,B 0,C 180,E1 24949.675,E2 24949.675} C_VEL
LIN {X 0,Y 532.617,Z 810.702,A -85,B 0,C 180,E1 24947.706,E2 24947.706} C_VEL
LIN {X 0,Y 531.394,Z 822.543,A -85,B 0,C 180,E1 24945.721,E2 24945.721} C_VEL
LIN {X 0,Y 530.407,Z 833.084,A -85,B 0,C 180,E1 24943.63,E2 24943.63} C_VEL
LIN {X 0,Y 529.678,Z 842.257,A -85,B 0,C 180,E1 24941.432,E2 24941.432} C_VEL
LIN {X 0,Y 529.164,Z 849.634,A -85,B 0,C 180,E1 24939.243,E2 24939.243} C_VEL
LIN {X 0,Y 528.84,Z 855.487,A -85,B 0,C 180,E1 24936.958,E2 24936.958} C_VEL
LIN {X 0,Y 528.68,Z 859.716,A -85,B 0,C 180,E1 24934.643,E2 24934.643} C_VEL
LIN {X 0,Y 528.594,Z 862.256,A -85,B 0,C 180,E1 24932.385,E2 24932.385} C_VEL
LIN {X 0,Y 528.581,Z 863.187,A -85,B 0,C 180,E1 24930.108,E2 24930.108} C_VEL
LIN {X 0,Y 528.591,Z 862.445,A -85,B 0,C 180,E1 24927.832,E2 24927.832} C_VEL
LIN {X 0,Y 528.671,Z 859.972,A -85,B 0,C 180,E1 24925.444,E2 24925.444} C_VEL
LIN {X 0,Y 528.832,Z 855.965,A -85,B 0,C 180,E1 24923.159,E2 24923.159} C_VEL
LIN {X 0,Y 529.123,Z 850.214,A -85,B 0,C 180,E1 24920.867,E2 24920.867} C_VEL
LIN {X 0,Y 529.621,Z 842.983,A -85,B 0,C 180,E1 24918.677,E2 24918.677} C_VEL
LIN {X 0,Y 530.326,Z 834.004,A -85,B 0,C 180,E1 24916.48,E2 24916.48} C_VEL
LIN {X 0,Y 531.287,Z 823.673,A -85,B 0,C 180,E1 24914.388,E2 24914.388} C_VEL
LIN {X 0,Y 532.563,Z 811.314,A -85,B 0,C 180,E1 24912.293,E2 24912.293} C_VEL
LIN {X 0,Y 534.073,Z 797.357,A -85,B 0,C 180,E1 24910.306,E2 24910.306} C_VEL
LIN {X 0,Y 535.744,Z 782.316,A -85,B 0,C 180,E1 24908.485,E2 24908.485} C_VEL
LIN {X 0,Y 537.581,Z 765.8,A -85,B 0,C 180,E1 24906.777,E2 24906.777} C_VEL
LIN {X 0,Y 539.546,Z 747.653,A -85,B 0,C 180,E1 24905.181,E2 24905.181} C_VEL
LIN {X 0,Y 541.418,Z 729.227,A -85,B 0,C 180,E1 24903.808,E2 24903.808} C_VEL
LIN {X 0,Y 543.211,Z 710.038,A -85,B 0,C 180,E1 24902.602,E2 24902.602} C_VEL
LIN {X 0,Y 544.933,Z 688.869,A -85,B 0,C 180,E1 24901.506,E2 24901.506} C_VEL
LIN {X 0,Y 546.395,Z 666.947,A -85,B 0,C 180,E1 24900.601,E2 24900.601} C_VEL
LIN {X 0,Y 547.5,Z 645.516,A -85,B 0,C 180,E1 24899.919,E2 24899.919} C_VEL
LIN {X 0,Y 548.585,Z 617.9,A -85,B 0,C 180,E1 24899.281,E2 24899.281} C_VEL
LIN {X 0,Y 552.911,Z 528.105,A -85,B 0,C 180,E1 24897.568,E2 24897.568} C_VEL
LIN {X 0,Y 556.199,Z 447.578,A -85,B 0,C 180,E1 24896.216,E2 24896.216} C_VEL
LIN {X 0,Y 558.848,Z 355.951,A -85,B 0,C 180,E1 24894.884,E2 24894.884} C_VEL
LIN {X 0,Y 560.858,Z 347.053,A -85,B 0,C 180,E1 24894.529,E2 24894.529} C_VEL
LIN {X 0,Y 560.927,Z 311.586,A -85,B 0,C 180,E1 24892.156,E2 24892.156} C_VEL
LIN {X 0,Y 561.314,Z 290.462,A -85,B 0,C 180,E1 24890.634,E2 24890.634} C_VEL
LIN {X 0,Y 552.958,Z 268.273,A -85,B 0,C 180,E1 24888.16,E2 24888.16} C_VEL
LIN {X 0,Y 544.509,Z 248.807,A -85,B 0,C 180,E1 24885.89,E2 24885.89} C_VEL
LIN {X 0,Y 536.433,Z 232.49,A -85,B 0,C 180,E1 24883.9,E2 24883.9} C_VEL
LIN {X 0,Y 531.595,Z 223.54,A -85,B 0,C 180,E1 24882.767,E2 24882.767} C_VEL
LIN {X 0,Y 529.865,Z 220.226,A -85,B 0,C 180,E1 24882.352,E2 24882.352} C_VEL
LIN {X 0,Y 529.686,Z 219.255,A -85,B 0,C 180,E1 24882.244,E2 24882.244} C_VEL
LIN {X 0,Y 529.667,Z 219.256,A -85,B 0,C 180,E1 24878.81,E2 24878.81} C_VEL
LIN {X 0,Y 529.684,Z 219.25,A -85,B 0,C 180,E1 24875.364,E2 24875.364} C_VEL
LIN {X 0,Y 529.678,Z 219.237,A -85,B 0,C 180,E1 24871.909,E2 24871.909} C_VEL
LIN {X 0,Y 529.675,Z 219.226,A -85,B 0,C 180,E1 24868.529,E2 24868.529} C_VEL
LIN {X 0,Y 529.676,Z 219.243,A -85,B 0,C 180,E1 24865.015,E2 24865.015} C_VEL
LIN {X 0,Y 529.677,Z 219.248,A -85,B 0,C 180,E1 24861.599,E2 24861.599} C_VEL
LIN {X 0,Y 529.679,Z 219.217,A -85,B 0,C 180,E1 24858.148,E2 24858.148} C_VEL
LIN {X 0,Y 529.678,Z 219.248,A -85,B 0,C 180,E1 24854.764,E2 24854.764} C_VEL
LIN {X 0,Y 529.673,Z 219.224,A -85,B 0,C 180,E1 24851.322,E2 24851.322} C_VEL
LIN {X 0,Y 529.669,Z 219.239,A -85,B 0,C 180,E1 24847.812,E2 24847.812} C_VEL
LIN {X 0,Y 529.678,Z 219.231,A -85,B 0,C 180,E1 24844.439,E2 24844.439} C_VEL
LIN {X 0,Y 529.686,Z 219.234,A -85,B 0,C 180,E1 24840.973,E2 24840.973} C_VEL
LIN {X 0,Y 529.66,Z 219.243,A -85,B 0,C 180,E1 24837.511,E2 24837.511} C_VEL
LIN {X 0,Y 529.674,Z 219.223,A -85,B 0,C 180,E1 24834.04,E2 24834.04} C_VEL
LIN {X 0,Y 529.685,Z 219.242,A -85,B 0,C 180,E1 24830.547,E2 24830.547} C_VEL
LIN {X 0,Y 529.667,Z 219.249,A -85,B 0,C 180,E1 24827.129,E2 24827.129} C_VEL
LIN {X 0,Y 529.655,Z 219.254,A -85,B 0,C 180,E1 24823.663,E2 24823.663} C_VEL
LIN {X 0,Y 529.687,Z 219.251,A -85,B 0,C 180,E1 24820.251,E2 24820.251} C_VEL
LIN {X 0,Y 529.678,Z 219.252,A -85,B 0,C 180,E1 24816.828,E2 24816.828} C_VEL
LIN {X 0,Y 529.649,Z 219.246,A -85,B 0,C 180,E1 24813.422,E2 24813.422} C_VEL
LIN {X 0,Y 529.683,Z 219.247,A -85,B 0,C 180,E1 24810.05,E2 24810.05} C_VEL
LIN {X 0,Y 529.677,Z 219.248,A -85,B 0,C 180,E1 24806.679,E2 24806.679} C_VEL
LIN {X 0,Y 529.66,Z 219.289,A -85,B 0,C 180,E1 24805.734,E2 24805.734} C_VEL
LIN {X 0,Y 530.757,Z 222.44,A -85,B 0,C 180,E1 24805.324,E2 24805.324} C_VEL
LIN {X 0,Y 532.266,Z 225.006,A -85,B 0,C 180,E1 24804.912,E2 24804.912} C_VEL
LIN {X 0,Y 540.989,Z 242.005,A -85,B 0,C 180,E1 24802.458,E2 24802.458} C_VEL
LIN {X 0,Y 551.488,Z 262.944,A -85,B 0,C 180,E1 24799.664,E2 24799.664} C_VEL
LIN {X 0,Y 563.478,Z 287.574,A -85,B 0,C 180,E1 24796.681,E2 24796.681} C_VEL
LIN {X 0,Y 567.952,Z 297.375,A -85,B 0,C 180,E1 24795.588,E2 24795.588} C_VEL
LIN {X 0,Y 566.382,Z 313.036,A -85,B 0,C 180,E1 24794.678,E2 24794.678} C_VEL
LIN {X 0,Y 569.212,Z 339.156,A -85,B 0,C 180,E1 24793.981,E2 24793.981} C_VEL
LIN {X 0,Y 561.49,Z 578.773,A -85,B 0,C 180,E1 24790.379,E2 24790.379} C_VEL
LIN {X 0,Y 558.297,Z 692.879,A -85,B 0,C 180,E1 24788.701,E2 24788.701} C_VEL
LIN {X 0,Y 556.902,Z 717.524,A -85,B 0,C 180,E1 24788.164,E2 24788.164} C_VEL
LIN {X 0,Y 555.258,Z 740.84,A -85,B 0,C 180,E1 24787.493,E2 24787.493} C_VEL
LIN {X 0,Y 553.211,Z 764.053,A -85,B 0,C 180,E1 24786.63,E2 24786.63} C_VEL
LIN {X 0,Y 550.987,Z 786.469,A -85,B 0,C 180,E1 24785.628,E2 24785.628} C_VEL
LIN {X 0,Y 548.466,Z 808.771,A -85,B 0,C 180,E1 24784.413,E2 24784.413} C_VEL
LIN {X 0,Y 545.954,Z 829.862,A -85,B 0,C 180,E1 24783.078,E2 24783.078} C_VEL
LIN {X 0,Y 543.365,Z 850.07,A -85,B 0,C 180,E1 24781.569,E2 24781.569} C_VEL
LIN {X 0,Y 540.876,Z 869.234,A -85,B 0,C 180,E1 24779.943,E2 24779.943} C_VEL
LIN {X 0,Y 538.406,Z 887.394,A -85,B 0,C 180,E1 24778.145,E2 24778.145} C_VEL
LIN {X 0,Y 536.191,Z 904.525,A -85,B 0,C 180,E1 24776.229,E2 24776.229} C_VEL
LIN {X 0,Y 534.175,Z 920.177,A -85,B 0,C 180,E1 24774.201,E2 24774.201} C_VEL
LIN {X 0,Y 532.465,Z 934.734,A -85,B 0,C 180,E1 24772.06,E2 24772.06} C_VEL
LIN {X 0,Y 531.024,Z 947.861,A -85,B 0,C 180,E1 24769.812,E2 24769.812} C_VEL
LIN {X 0,Y 529.956,Z 959.277,A -85,B 0,C 180,E1 24767.57,E2 24767.57} C_VEL
LIN {X 0,Y 529.085,Z 970.28,A -85,B 0,C 180,E1 24765.005,E2 24765.005} C_VEL
LIN {X 0,Y 528.596,Z 978.281,A -85,B 0,C 180,E1 24762.786,E2 24762.786} C_VEL
LIN {X 0,Y 528.245,Z 986.314,A -85,B 0,C 180,E1 24760.029,E2 24760.029} C_VEL
LIN {X 0,Y 528.098,Z 991.25,A -85,B 0,C 180,E1 24757.835,E2 24757.835} C_VEL
LIN {X 0,Y 528.05,Z 995.309,A -85,B 0,C 180,E1 24755.433,E2 24755.433} C_VEL
LIN {X 0,Y 528.058,Z 997.854,A -85,B 0,C 180,E1 24752.93,E2 24752.93} C_VEL
LIN {X 0,Y 528.073,Z 998.814,A -85,B 0,C 180,E1 24750.759,E2 24750.759} C_VEL
LIN {X 0,Y 528.091,Z 998.55,A -85,B 0,C 180,E1 24748.372,E2 24748.372} C_VEL
LIN {X 0,Y 528.095,Z 996.5,A -85,B 0,C 180,E1 24745.765,E2 24745.765} C_VEL
LIN {X 0,Y 528.112,Z 993.292,A -85,B 0,C 180,E1 24743.477,E2 24743.477} C_VEL
LIN {X 0,Y 528.202,Z 987.95,A -85,B 0,C 180,E1 24740.85,E2 24740.85} C_VEL
LIN {X 0,Y 528.409,Z 981.754,A -85,B 0,C 180,E1 24738.579,E2 24738.579} C_VEL
LIN {X 0,Y 528.804,Z 973.873,A -85,B 0,C 180,E1 24736.217,E2 24736.217} C_VEL
LIN {X 0,Y 529.458,Z 963.843,A -85,B 0,C 180,E1 24733.77,E2 24733.77} C_VEL
LIN {X 0,Y 530.258,Z 953.621,A -85,B 0,C 180,E1 24731.645,E2 24731.645} C_VEL
LIN {X 0,Y 531.541,Z 939.728,A -85,B 0,C 180,E1 24729.174,E2 24729.174} C_VEL
LIN {X 0,Y 532.919,Z 926.263,A -85,B 0,C 180,E1 24727.109,E2 24727.109} C_VEL
LIN {X 0,Y 534.753,Z 909.549,A -85,B 0,C 180,E1 24724.884,E2 24724.884} C_VEL
LIN {X 0,Y 536.55,Z 894.005,A -85,B 0,C 180,E1 24723.074,E2 24723.074} C_VEL
LIN {X 0,Y 538.909,Z 873.935,A -85,B 0,C 180,E1 24721.036,E2 24721.036} C_VEL
LIN {X 0,Y 541.194,Z 854.701,A -85,B 0,C 180,E1 24719.341,E2 24719.341} C_VEL
LIN {X 0,Y 543.603,Z 833.893,A -85,B 0,C 180,E1 24717.763,E2 24717.763} C_VEL
LIN {X 0,Y 545.862,Z 813.459,A -85,B 0,C 180,E1 24716.414,E2 24716.414} C_VEL
LIN {X 0,Y 548.077,Z 791.418,A -85,B 0,C 180,E1 24715.178,E2 24715.178} C_VEL
LIN {X 0,Y 550.284,Z 768.641,A -85,B 0,C 180,E1 24714.098,E2 24714.098} C_VEL
LIN {X 0,Y 552.167,Z 745.38,A -85,B 0,C 180,E1 24713.206,E2 24713.206} C_VEL
LIN {X 0,Y 553.867,Z 721.472,A -85,B 0,C 180,E1 24712.47,E2 24712.47} C_VEL
LIN {X 0,Y 555.081,Z 698.627,A -85,B 0,C 180,E1 24711.945,E2 24711.945} C_VEL
LIN {X 0,Y 556.026,Z 670.252,A -85,B 0,C 180,E1 24711.484,E2 24711.484} C_VEL
LIN {X 0,Y 558.703,Z 568.517,A -85,B 0,C 180,E1 24709.989,E2 24709.989} C_VEL
LIN {X 0,Y 562.298,Z 475.68,A -85,B 0,C 180,E1 24708.47,E2 24708.47} C_VEL
